// TwinCAT 3 PLC project Rohlik_Expansion
// ProgramVersion: 3.1.4024.0
// libraries:
//   CmpBitmapPool, * (System)
//   Tc2_EtherCAT, * (Beckhoff Automation GmbH)
//   Tc2_IoFunctions, * (Beckhoff Automation GmbH)
//   Tc2_MC2, * (Beckhoff Automation GmbH)
//   Tc2_ModbusSrv, * (Beckhoff Automation GmbH)
//   Tc2_Standard, * (Beckhoff Automation GmbH)
//   Tc2_SUPS, * (Beckhoff Automation GmbH)
//   Tc2_System, * (Beckhoff Automation GmbH)
//   Tc2_Utilities, * (Beckhoff Automation GmbH)
//   Tc3_Module, * (Beckhoff Automation GmbH)
//   Tc3_PackML_V2, * (Beckhoff Automation GmbH)
//   Util, * (System)
//   VisuDialogs, * (System)
// project tree:
//   02DUTs/ E_PMLUserUnitMode.TcDUT (not stored), E_UnitName.TcDUT (not stored), ModuleID.TcDUT, ST_ChangeIntoProduction.TcDUT, ST_UnitInfo.TcDUT (not stored)
//   Ads/ AbortToteRequestParams.TcDUT (not stored), AutostoreControlCommand.TcDUT, BarcodeValidationRequestParams.TcDUT (not stored), BarcodeVerificationResult.TcDUT (not stored), ButtonStatus.TcDUT (not stored), AirPressureStatus.TcDUT (not stored), DigitalInputStatus.TcDUT (not stored), DigitalOutputStatus.TcDUT, EStopStatus.TcDUT, E_SAFETYDOOR.TcDUT, E_SafetyStates.TcDUT (not stored), FB_AirPressure_Subsystem.TcPOU (not stored), FB_HeartBeat_Subsystem.TcPOU (not stored), FB_Light_tower_module.TcPOU (not stored), FB_MachineControl_Subsystem.TcPOU, FB_Safety_Subsystem.TcPOU, FB_Tote_Subsystem.TcPOU, GeneralStatus.TcDUT, HeartbeatParams.TcDUT (not stored), InboundToteParams.TcDUT, InitToteRequestParams.TcDUT (not stored), LightCurtainStatus.TcDUT, MachineCommandStructure.TcDUT (not stored), MachineControlCommand.TcDUT, MachineControlCommand_1.TcDUT, MachineStatus.TcDUT (not stored), MethodCallReturnValue.TcDUT (not stored), ModelIdentifier.TcDUT (not stored), OrderToteCommand.TcDUT (not stored), OutboundToteParams.TcDUT, PerturbToteParams.TcDUT (not stored), SafetyDoorStatus.TcDUT, SafetyStatus.TcDUT (not stored), SensorStatus.TcDUT, StationMode.TcDUT (not stored), ST_BagOpen.TcDUT, ST_LightTower.TcDUT (not stored), SwapToteParams.TcDUT (not stored), ToteData.TcPOU (not stored), UpdateLightTowerParams.TcDUT, UpdateStationModeParams.TcDUT (not stored)
//   Ads/Ads/ BagOpeningStatus.TcPOU, ST_LightTowerAction.TcDUT (not stored)
//   GVLs/ GVL.TcGVL, GVL_SAFETY.TcGVL (not stored), G_HMI.TcGVL, G_IO.TcGVL, ST_Ifm_Qualifier.TcDUT (not stored), ST_Ifm_RX.TcDUT (not stored), ST_Ifm_TX.TcDUT (not stored), ST_IO_16.TcDUT (not stored), ST_SafetyIO.TcDUT (not stored)
//   / EtherCAT_Task.TcTTO, GlobalTextList.TcGTLO, MianTask.TcTTO (not stored), VisualizationManager.TcVMO (not stored), VISU_TASK.TcTTO (not stored)
//   LogTECH/ LogTechControlCmd.TcDUT (not stored), LogTechStatus.TcDUT, LogTechTransferStatus.TcDUT
//   Mian/axis/ AxisHMI_Ex.TcVIS (not stored), E_HomingSteps.TcDUT (not stored), FB_MotionAxis_MC.TcPOU (not stored), MC_HomeAxis.TcPOU (not stored), ST_MotionAxis_MC.TcDUT
//   Mian/DUTs/ BagStatus.TcDUT (not stored), Buffer_roller.TcDUT, E_Condition.TcDUT, E_LoadingStates.TcDUT, E_SampleStates.TcDUT, E_RollerStates.TcDUT (not stored), E_AutoStore_States.TcDUT, E_topic_sample.TcDUT (not stored), E_Transfer.TcDUT (not stored), E_WorkingStates.TcDUT (not stored), FB_DigitalInput.TcPOU (not stored), FB_GPWM.TcPOU (not stored), Inbound.TcDUT, I_Common.TcIO (not stored), OrderToteErrorStatus.TcDUT (not stored), Outbound.TcDUT, Prepare_Date_Time.TcPOU (not stored), Roller.TcDUT (not stored), Roller_x.TcDUT (not stored), Roller_y.TcDUT, ServerityLevelType.TcDUT, ST_Alarm_Hmi.TcDUT (not stored), ST_control_pannel.TcDUT, ST_EVENT.TcDUT (not stored), ST_safetyDoor.TcDUT (not stored), ToteStatus.TcDUT (not stored), ToteSubsystemWorkflowStatus.TcDUT, Valve.TcDUT (not stored)
//   Mian/ FB_Generic.TcPOU (not stored), FB_Machine.TcPOU, FB_mcp.TcPOU (not stored), FB_Sample.TcPOU (not stored), FB_loading_tote.TcPOU (not stored), FB_autoStore.TcPOU, FB_StateMachine.TcPOU, FB_working_tote.TcPOU, FB_Visu.TcPOU (not stored), FB_WriteLog.TcPOU (not stored), MAIN.TcPOU
//   PubSub/ E_Topics.TcDUT, I_PubSubService.TcIO (not stored), I_SubCallback.TcIO (not stored), KeyAndValue.TcDUT, PubSubData.TcDUT (not stored), PubSubService.TcPOU, ST_TracePublish.TcDUT (not stored), SubscriberCell.TcDUT
//   VISUs/ ImagePool.TcIPO (not stored), visu_main.TcVIS (not stored)
//   VISUs/Templates/ visu_autoStore.TcVIS, VIS_TemplateCommand.TcVIS (not stored), VIS_TemplateKeys.TcVIS (not stored), VIS_TemplateMachine.TcVIS (not stored), VIS_TemplatePMLStateModel.TcVIS, VIS_TemplateToProduction.TcVIS (not stored), v_io_autoStore.TcVIS
//   VISUs/VISUs/ Menu.TcVIS (not stored), visu_2sys.TcVIS, visu_loading.TcVIS (not stored), visu_operation.TcVIS, visu_sample.TcVIS (not stored), visu_manual.TcVIS, visu_working1.TcVIS, visu_autoStore1.TcVIS, visu_working2.TcVIS, v_alarm.TcVIS, v_io_loading.TcVIS (not stored), v_io_working1.TcVIS, v_io_working2.TcVIS (not stored)
// real-time tasks:
//   TASK PlcTask: cycle T#4ms, priority 20, ADS port 350
//   TASK EtherCAT_Task: cycle T#2ms, priority 2, ADS port 351
//   TASK VISU_TASK: cycle T#100000us, priority 30, ADS port 352
// motion (NC):
//   TASK NC-Task 1 SAF: cycle T#2ms, priority 4, ADS port 501
//   TASK NC-Task 1 SVB: cycle T#10ms, priority 8, ADS port 511
//   AXIS lift_motor (id 3)
//     Velo: SlowManual=5, FastManual=20
//     PositionAreaControl: Enable=false
//     OtherSettings: AllowMotionCmdToSlave=true
//     encoder EncType=19
//       EncPara: ScaleFactorNumerator=3.333333333333, ScaleFactorDenominator=8388608, Inverse=true, MaxCount=#xffffffff, ReferenceSystem=1
//         SoftEndMinControl: Enable=true, Range=-5
//         SoftEndMaxControl: Enable=true, Range=800
//         Inc: RefSoftSyncMask=#x00800000
//     drive DrvType=16
//       DrvPara: Inverse=true, MaxCount=#xffffffff, DriveControlDWord=#x00020100
//         Analog: TorqueSetpointScale=10, ScaleFactorActTorque=0.1
//         TimeComp: TaskDelayCycles=1
//     controller CtrType=1
//       CtrPara: PriorControlFactor=1
//         PosDiffControl: Enable=false
//         Observer: BandWidth=20
//   AXIS working1_lift_motor (id 4)
//     PositionAreaControl: Enable=false
//     OtherSettings: AllowMotionCmdToSlave=true
//     encoder EncType=19
//       EncPara: ScaleFactorNumerator=5, ScaleFactorDenominator=8388608, Inverse=true, MaxCount=#xffffffff, ReferenceSystem=1
//         SoftEndMinControl: Enable=true, Range=-5
//         SoftEndMaxControl: Enable=true, Range=140
//         Inc: RefSoftSyncMask=#x00800000
//     drive DrvType=16
//       DrvPara: Inverse=true, MaxCount=#xffffffff, DriveControlDWord=#x00020100
//         Analog: TorqueSetpointScale=10, ScaleFactorActTorque=0.1
//         TimeComp: TaskDelayCycles=1
//     controller CtrType=1
//       CtrPara: PriorControlFactor=1
//         PosDiffControl: Enable=false
//         Observer: BandWidth=20
//   AXIS working1_open_bag (id 5)
//     General: UnitName=°
//     Dynamic: Acceleration=75, Deceleration=75, Jerk=112.5
//     Velo: SlowManual=1, FastManual=5, Maximum=300
//     PositionAreaControl: Enable=false
//     OtherSettings: AllowMotionCmdToSlave=true
//     encoder EncType=19
//       EncPara: ScaleFactorNumerator=36, ScaleFactorDenominator=8388608, MaxCount=#xffffffff, ReferenceSystem=1
//         SoftEndMinControl: Enable=true
//         SoftEndMaxControl: Enable=true, Range=56
//         Inc: RefSoftSyncMask=#x00800000
//     drive DrvType=16
//       DrvPara: MaxCount=#xffffffff, DriveControlDWord=#x00020100
//         Analog: TorqueSetpointScale=10, ScaleFactorActTorque=0.1
//         TimeComp: TaskDelayCycles=1
//     controller CtrType=1
//       CtrPara: PriorControlFactor=1
//         PosDiffControl: Enable=false
//         Observer: BandWidth=20
//   AXIS working2_lift_motor (id 1)
//     PositionAreaControl: Enable=false
//     OtherSettings: AllowMotionCmdToSlave=true
//     encoder EncType=19
//       EncPara: ScaleFactorNumerator=5, ScaleFactorDenominator=8388608, Inverse=true, MaxCount=#xffffffff, ReferenceSystem=1
//         SoftEndMinControl: Enable=true, Range=-5
//         SoftEndMaxControl: Enable=true, Range=140
//         Inc: RefSoftSyncMask=#x00800000
//     drive DrvType=16
//       DrvPara: Inverse=true, MaxCount=#xffffffff, DriveControlDWord=#x00020100
//         Analog: TorqueSetpointScale=10, ScaleFactorActTorque=0.1
//         TimeComp: TaskDelayCycles=1
//     controller CtrType=1
//       CtrPara: PriorControlFactor=1
//         PosDiffControl: Enable=false
//         Observer: BandWidth=20
//   AXIS working2_open_bag (id 2)
//     General: UnitName=°
//     Dynamic: Acceleration=75, Deceleration=75, Jerk=112.5
//     Velo: Maximum=300
//     PositionAreaControl: Enable=false
//     OtherSettings: AllowMotionCmdToSlave=true
//     encoder EncType=19
//       EncPara: ScaleFactorNumerator=36, ScaleFactorDenominator=8388608, MaxCount=#xffffffff, ReferenceSystem=1
//         SoftEndMinControl: Enable=true
//         SoftEndMaxControl: Enable=true, Range=56
//         Inc: RefSoftSyncMask=#x00800000
//     drive DrvType=16
//       DrvPara: MaxCount=#xffffffff, DriveControlDWord=#x00020100
//         Analog: TorqueSetpointScale=10, ScaleFactorActTorque=0.1
//         TimeComp: TaskDelayCycles=1
//     controller CtrType=1
//       CtrPara: PriorControlFactor=1
//         PosDiffControl: Enable=false
//         Observer: BandWidth=20
//   AXIS autostore1_transfer (id 6)
//     OtherSettings: AllowMotionCmdToSlave=true
//     encoder EncType=1
//     drive DrvType=5
//       Analog: TorqueSetpointScale=10, ScaleFactorActTorque=0.1
//     controller CtrType=1
//       CtrPara: PriorControlFactor=1
//         Observer: BandWidth=20
//   AXIS autostore1_lift (id 7)
//     OtherSettings: AllowMotionCmdToSlave=true
//     encoder EncType=1
//     drive DrvType=5
//       Analog: TorqueSetpointScale=10, ScaleFactorActTorque=0.1
//     controller CtrType=1
//       CtrPara: PriorControlFactor=1
//         Observer: BandWidth=20
//   AXIS autostore2_transfer (id 8)
//     OtherSettings: AllowMotionCmdToSlave=true
//     encoder EncType=1
//     drive DrvType=5
//       Analog: TorqueSetpointScale=10, ScaleFactorActTorque=0.1
//     controller CtrType=1
//       CtrPara: PriorControlFactor=1
//         Observer: BandWidth=20
//   AXIS autostore2_lift (id 9)
//     OtherSettings: AllowMotionCmdToSlave=true
//     encoder EncType=1
//     drive DrvType=5
//       Analog: TorqueSetpointScale=10, ScaleFactorActTorque=0.1
//     controller CtrType=1
//       CtrPara: PriorControlFactor=1
//         Observer: BandWidth=20
// I/O:
//   DEVICE Device 2 (RT-Ethernet Adapter)
//   DEVICE MCP, AmsNetId 192.168.17.27.4.1
//     Box 1 (CU2508) [CU2508 Ethernet Port]
//     MCP-EK1100 [EK1100 EtherCAT Coupler (2A E-Bus)]
//       DI0 [EL1809 16Ch. Dig. Input 24V, 3ms]
//       DI1 [EL1809 16Ch. Dig. Input 24V, 3ms]
//       DO0 [EL2809 16Ch. Dig. Output 24V, 0.5A]
//       DO1 [EL2809 16Ch. Dig. Output 24V, 0.5A]
//       Term 7 (EL6910) [EL6910, TwinSAFE PLC]
//       SI0 [EL1904, 4 Ch. Safety Input 24V, TwinSAFE]
//         modules: Module 1 (FSOES)
//       SI1 [EL1904, 4 Ch. Safety Input 24V, TwinSAFE]
//         modules: Module 1 (FSOES)
//       SI2 [EL1904, 4 Ch. Safety Input 24V, TwinSAFE]
//         modules: Module 1 (FSOES)
//       SI3 [EL1904, 4 Ch. Safety Input 24V, TwinSAFE]
//         modules: Module 1 (FSOES)
//       SO0 [EL2904, 4 Ch. Safety Output 24V, 0.5A, TwinSAFE]
//         modules: Module 1 (FSOES), Module 2 (DO)
//       SO4 [EL2904, 4 Ch. Safety Output 24V, 0.5A, TwinSAFE]
//         modules: Module 1 (FSOES), Module 2 (DO)
//       Term 50 (EL9410) [EL9410 E-Bus Power Supplier  (Diagnostics)]
//       Term 13 (EL3064) [EL3064 4Ch. Ana. Input 0-10V]
//       SI7 [EL1904, 4 Ch. Safety Input 24V, TwinSAFE]
//         modules: Module 1 (FSOES)
//       SI8 [EL1904, 4 Ch. Safety Input 24V, TwinSAFE]
//         modules: Module 1 (FSOES)
//       SO5 [EL2904, 4 Ch. Safety Output 24V, 0.5A, TwinSAFE]
//         modules: Module 1 (FSOES), Module 2 (DO)
//       SO6 [EL2904, 4 Ch. Safety Output 24V, 0.5A, TwinSAFE]
//         modules: Module 1 (FSOES), Module 2 (DO)
//       Term 14 (EL6631-0010) [EL6631-0010 PROFINET IO Device]
//       Term 15 (EL9011) [EL9011 End Terminal]
//   DEVICE Lift, AmsNetId 192.168.17.27.5.1
//     Box 16 (CU2508) [CU2508 Ethernet Port]
//     Term 17 (EK1100) [EK1100 EtherCAT Coupler (2A E-Bus)]
//       DI2 [EL1809 16Ch. Dig. Input 24V, 3ms]
//       DI3 [EL1809 16Ch. Dig. Input 24V, 3ms]
//       DO2 [EL2809 16Ch. Dig. Output 24V, 0.5A]
//       DO3 [EL2809 16Ch. Dig. Output 24V, 0.5A]
//       SI4 [EL1904, 4 Ch. Safety Input 24V, TwinSAFE]
//         modules: Module 1 (FSOES)
//       SI5 [EL1904, 4 Ch. Safety Input 24V, TwinSAFE]
//         modules: Module 1 (FSOES)
//       SI6 [EL1904, 4 Ch. Safety Input 24V, TwinSAFE]
//         modules: Module 1 (FSOES)
//       SO1 [EL2904, 4 Ch. Safety Output 24V, 0.5A, TwinSAFE]
//         modules: Module 1 (FSOES), Module 2 (DO)
//       Term 10 (EL9011) [EL9011 End Terminal]
//     lift_lift [SV660_1Axis_00915]
//     Box 26 (ifm IO-Link Master AL1332) [ifm IO-Link Master AL1332]
//       modules: Module 1 (IOL_4/4_I/O-Bytes), Module 2 (IOL_4/4_I/O-Bytes), Module 3 (IOL_4/4_I/O-Bytes), Module 4 (IOL_4/4_I/O-Bytes), Module 5 (IOL_4/4_I/O-Bytes), Module 6 (IOL_4/4_I/O-Bytes), Module 7 (IOL_4/4_I/O-Bytes), Module 8 (IOL_4/4_I/O-Bytes)
//   DEVICE Place1, AmsNetId 192.168.17.27.6.1
//     Box 26 (CU2508) [CU2508 Ethernet Port]
//     Term 27 (EK1100) [EK1100 EtherCAT Coupler (2A E-Bus)]
//       DI4 [EL1809 16Ch. Dig. Input 24V, 3ms]
//       DI5 [EL1809 16Ch. Dig. Input 24V, 3ms]
//       DO4 [EL2809 16Ch. Dig. Output 24V, 0.5A]
//       SO2 [EL2904, 4 Ch. Safety Output 24V, 0.5A, TwinSAFE]
//         modules: Module 1 (FSOES), Module 2 (DO)
//       Term 53 (EL9410) [EL9410 E-Bus Power Supplier  (Diagnostics)]
//       DO6 [EL2809 16Ch. Dig. Output 24V, 0.5A]
//       Term 9 (EL9011) [EL9011 End Terminal]
//     place1_lift [SV660_1Axis_00915]
//     place_openbag [SV660_1Axis_00915]
//     Box 36 (ifm IO-Link Master AL1332) [ifm IO-Link Master AL1332]
//       modules: Module 1 (IOL_4/4_I/O-Bytes), Module 2 (IOL_4/4_I/O-Bytes), Module 3 (IOL_4/4_I/O-Bytes), Module 4 (IOL_4/4_I/O-Bytes), Module 5 (IOL_4/4_I/O-Bytes), Module 6 (IOL_4/4_I/O-Bytes), Module 7 (IOL_4/4_I/O-Bytes), Module 8 (IOL_4/4_I/O-Bytes)
//   DEVICE Place2, AmsNetId 192.168.17.27.7.1
//     Box 35 (CU2508) [CU2508 Ethernet Port]
//     Term 36 (EK1100) [EK1100 EtherCAT Coupler (2A E-Bus)]
//       DI6 [EL1809 16Ch. Dig. Input 24V, 3ms]
//       DI7 [EL1809 16Ch. Dig. Input 24V, 3ms]
//       DO5 [EL2809 16Ch. Dig. Output 24V, 0.5A]
//       SO3 [EL2904, 4 Ch. Safety Output 24V, 0.5A, TwinSAFE]
//         modules: Module 1 (FSOES), Module 2 (DO)
//       Term 51 (EL9410) [EL9410 E-Bus Power Supplier  (Diagnostics)]
//       DO7 [EL2809 16Ch. Dig. Output 24V, 0.5A]
//       Term 9 (EL9011) [EL9011 End Terminal]
//     place2_lift [SV660_1Axis_00915]
//     place2_openbag [SV660_1Axis_00915]
//     Box 46 (ifm IO-Link Master AL1332) [ifm IO-Link Master AL1332]
//       modules: Module 1 (IOL_4/4_I/O-Bytes), Module 2 (IOL_4/4_I/O-Bytes), Module 3 (IOL_4/4_I/O-Bytes), Module 4 (IOL_4/4_I/O-Bytes), Module 5 (IOL_4/4_I/O-Bytes), Module 6 (IOL_4/4_I/O-Bytes), Module 7 (IOL_4/4_I/O-Bytes), Module 8 (IOL_4/4_I/O-Bytes)
//   DEVICE Device 1 (EtherCAT Automation Protocol), AmsNetId 192.168.11.159.2.1
// variable links:
//   Lift <-> MCP/MCP-EK1100/Term 7 (EL6910)
//     Term 17 (EK1100)/SI5/Module 1 (FSOES)/RxPDO/FSOE <-> ConnectionInputs/Message_29 TxPDO
//     Term 17 (EK1100)/SI6/Module 1 (FSOES)/RxPDO/FSOE <-> ConnectionInputs/Message_30 TxPDO
//     Term 17 (EK1100)/SI5/Module 1 (FSOES)/TxPDO/FSOE <-> ConnectionOutputs/Message_29 RxPDO
//     Term 17 (EK1100)/SI6/Module 1 (FSOES)/TxPDO/FSOE <-> ConnectionOutputs/Message_30 RxPDO
//   MCP <-> Lift/Term 17 (EK1100)/SI4
//     MCP-EK1100/Term 7 (EL6910)/ConnectionInputs/Message_28 TxPDO <-> Module 1 (FSOES)/RxPDO/FSOE
//     MCP-EK1100/Term 7 (EL6910)/ConnectionOutputs/Message_28 RxPDO <-> Module 1 (FSOES)/TxPDO/FSOE
//   MCP <-> Lift/Term 17 (EK1100)/SO1
//     MCP-EK1100/Term 7 (EL6910)/ConnectionInputs/Message_31 TxPDO <-> Module 1 (FSOES)/RxPDO/FSOE
//     MCP-EK1100/Term 7 (EL6910)/ConnectionOutputs/Message_31 RxPDO <-> Module 1 (FSOES)/TxPDO/FSOE
//   MCP <-> MCP/MCP-EK1100/SI0
//     MCP-EK1100/Term 7 (EL6910)/ConnectionOutputs/Message_22 RxPDO <-> Module 1 (FSOES)/TxPDO/FSOE
//   MCP <-> MCP/MCP-EK1100/SI1
//     MCP-EK1100/Term 7 (EL6910)/ConnectionInputs/Message_23 TxPDO <-> Module 1 (FSOES)/RxPDO/FSOE
//   MCP <-> MCP/MCP-EK1100/SI2
//     MCP-EK1100/Term 7 (EL6910)/ConnectionInputs/Message_24 TxPDO <-> Module 1 (FSOES)/RxPDO/FSOE
//     MCP-EK1100/Term 7 (EL6910)/ConnectionOutputs/Message_24 RxPDO <-> Module 1 (FSOES)/TxPDO/FSOE
//   MCP <-> MCP/MCP-EK1100/SI3
//     MCP-EK1100/Term 7 (EL6910)/ConnectionInputs/Message_27 TxPDO <-> Module 1 (FSOES)/RxPDO/FSOE
//   MCP <-> MCP/MCP-EK1100/SO0
//     MCP-EK1100/Term 7 (EL6910)/ConnectionInputs/Message_26 TxPDO <-> Module 1 (FSOES)/RxPDO/FSOE
//   MCP <-> MCP/MCP-EK1100/SO4
//     MCP-EK1100/Term 7 (EL6910)/ConnectionInputs/Message_36 TxPDO <-> Module 1 (FSOES)/RxPDO/FSOE
//   MCP <-> MCP/MCP-EK1100/SO6
//     MCP-EK1100/Term 7 (EL6910)/ConnectionInputs/Message_72 TxPDO <-> Module 1 (FSOES)/RxPDO/FSOE
//     MCP-EK1100/Term 7 (EL6910)/ConnectionOutputs/Message_72 RxPDO <-> Module 1 (FSOES)/TxPDO/FSOE
//   MCP <-> MCP/MCP-EK1100/Term 7 (EL6910)
//     MCP-EK1100/SI0/Module 1 (FSOES)/RxPDO/FSOE <-> ConnectionInputs/Message_22 TxPDO
//     MCP-EK1100/SI1/Module 1 (FSOES)/TxPDO/FSOE <-> ConnectionOutputs/Message_23 RxPDO
//     MCP-EK1100/SI3/Module 1 (FSOES)/TxPDO/FSOE <-> ConnectionOutputs/Message_27 RxPDO
//     MCP-EK1100/SO0/Module 1 (FSOES)/TxPDO/FSOE <-> ConnectionOutputs/Message_26 RxPDO
//     MCP-EK1100/SO4/Module 1 (FSOES)/TxPDO/FSOE <-> ConnectionOutputs/Message_36 RxPDO
//     MCP-EK1100/SO5/Module 1 (FSOES)/TxPDO/FSOE <-> ConnectionOutputs/Message_71 RxPDO
//     MCP-EK1100/SO5/Module 1 (FSOES)/RxPDO/FSOE <-> ConnectionInputs/Message_71 TxPDO
//   MCP <-> Place2/Term 36 (EK1100)/SO3
//     MCP-EK1100/Term 7 (EL6910)/ConnectionInputs/Message_33 TxPDO <-> Module 1 (FSOES)/RxPDO/FSOE
//     MCP-EK1100/Term 7 (EL6910)/ConnectionOutputs/Message_33 RxPDO <-> Module 1 (FSOES)/TxPDO/FSOE
//   Place1 <-> MCP/MCP-EK1100/Term 7 (EL6910)
//     Term 27 (EK1100)/SO2/Module 1 (FSOES)/RxPDO/FSOE <-> ConnectionInputs/Message_32 TxPDO
//     Term 27 (EK1100)/SO2/Module 1 (FSOES)/TxPDO/FSOE <-> ConnectionOutputs/Message_32 RxPDO
//   NC-Task 1 SAF/Axes/lift_motor <-> Lift/lift_lift
//     Drive/Inputs/In/nDataIn1 <-> Inputs/Following error actual value
//     Drive/Inputs/In/nDataIn3[0] <-> Inputs/Torque actual value
//     Drive/Inputs/In/nDcOutputTime <-> InfoData/DcOutputShift
//     Drive/Inputs/In/nState1 <-> Inputs/Statusword
//     Drive/Inputs/In/nState2 <-> Inputs/Statusword @bit 8
//     Drive/Inputs/In/nState4 @bit 1 <-> WcState/InputToggle
//     Drive/Inputs/In/nState4 <-> WcState/WcState
//     Drive/Outputs/Out/nCtrl1 <-> Outputs/Controlword
//     Drive/Outputs/Out/nCtrl2 <-> Outputs/Controlword @bit 8
//     Drive/Outputs/Out/nDataOut1 <-> Outputs/Target position
//     Enc/Inputs/In/nDataIn1 <-> Inputs/Position actual value
//     Enc/Inputs/In/nDataIn3 <-> Inputs/Touch probe pos1 pos value
//     Enc/Inputs/In/nDataIn5 <-> Inputs/Touch probe pos2 pos value
//     Enc/Inputs/In/nDcInputTime <-> InfoData/DcInputShift
//     Enc/Inputs/In/nState4 @bit 1 <-> WcState/InputToggle
//     Enc/Inputs/In/nState4 <-> WcState/WcState
//     Enc/Inputs/In/nState5 <-> Inputs/Touch probe status
//     Enc/Inputs/In/nState6 <-> Inputs/Touch probe status @bit 8
//     Enc/Outputs/Out/nCtrl5 <-> Outputs/Touch probe function
//     Enc/Outputs/Out/nCtrl6 <-> Outputs/Touch probe function @bit 8
//   NC-Task 1 SAF/Axes/working1_lift_motor <-> Place1/place1_lift
//     Drive/Inputs/In/nDataIn1 <-> Inputs/Following error actual value
//     Drive/Inputs/In/nDataIn3[0] <-> Inputs/Torque actual value
//     Drive/Inputs/In/nDcOutputTime <-> InfoData/DcOutputShift
//     Drive/Inputs/In/nState1 <-> Inputs/Statusword
//     Drive/Inputs/In/nState2 <-> Inputs/Statusword @bit 8
//     Drive/Inputs/In/nState4 @bit 1 <-> WcState/InputToggle
//     Drive/Inputs/In/nState4 <-> WcState/WcState
//     Drive/Outputs/Out/nCtrl1 <-> Outputs/Controlword
//     Drive/Outputs/Out/nCtrl2 <-> Outputs/Controlword @bit 8
//     Drive/Outputs/Out/nDataOut1 <-> Outputs/Target position
//     Enc/Inputs/In/nDataIn1 <-> Inputs/Position actual value
//     Enc/Inputs/In/nDataIn3 <-> Inputs/Touch probe pos1 pos value
//     Enc/Inputs/In/nDataIn5 <-> Inputs/Touch probe pos2 pos value
//     Enc/Inputs/In/nDcInputTime <-> InfoData/DcInputShift
//     Enc/Inputs/In/nState4 @bit 1 <-> WcState/InputToggle
//     Enc/Inputs/In/nState4 <-> WcState/WcState
//     Enc/Inputs/In/nState5 <-> Inputs/Touch probe status
//     Enc/Inputs/In/nState6 <-> Inputs/Touch probe status @bit 8
//     Enc/Outputs/Out/nCtrl5 <-> Outputs/Touch probe function
//     Enc/Outputs/Out/nCtrl6 <-> Outputs/Touch probe function @bit 8
//   NC-Task 1 SAF/Axes/working1_open_bag <-> Place1/place_openbag
//     Drive/Inputs/In/nDataIn1 <-> Inputs/Following error actual value
//     Drive/Inputs/In/nDataIn3[0] <-> Inputs/Torque actual value
//     Drive/Inputs/In/nDcOutputTime <-> InfoData/DcOutputShift
//     Drive/Inputs/In/nState1 <-> Inputs/Statusword
//     Drive/Inputs/In/nState2 <-> Inputs/Statusword @bit 8
//     Drive/Inputs/In/nState4 @bit 1 <-> WcState/InputToggle
//     Drive/Inputs/In/nState4 <-> WcState/WcState
//     Drive/Outputs/Out/nCtrl1 <-> Outputs/Controlword
//     Drive/Outputs/Out/nCtrl2 <-> Outputs/Controlword @bit 8
//     Drive/Outputs/Out/nDataOut1 <-> Outputs/Target position
//     Enc/Inputs/In/nDataIn1 <-> Inputs/Position actual value
//     Enc/Inputs/In/nDataIn3 <-> Inputs/Touch probe pos1 pos value
//     Enc/Inputs/In/nDataIn5 <-> Inputs/Touch probe pos2 pos value
//     Enc/Inputs/In/nDcInputTime <-> InfoData/DcInputShift
//     Enc/Inputs/In/nState4 @bit 1 <-> WcState/InputToggle
//     Enc/Inputs/In/nState4 <-> WcState/WcState
//     Enc/Inputs/In/nState5 <-> Inputs/Touch probe status
//     Enc/Inputs/In/nState6 <-> Inputs/Touch probe status @bit 8
//     Enc/Outputs/Out/nCtrl5 <-> Outputs/Touch probe function
//     Enc/Outputs/Out/nCtrl6 <-> Outputs/Touch probe function @bit 8
//   NC-Task 1 SAF/Axes/working2_lift_motor <-> Place2/place2_lift
//     Drive/Inputs/In/nDataIn1 <-> Inputs/Following error actual value
//     Drive/Inputs/In/nDataIn3[0] <-> Inputs/Torque actual value
//     Drive/Inputs/In/nDcOutputTime <-> InfoData/DcOutputShift
//     Drive/Inputs/In/nState1 <-> Inputs/Statusword
//     Drive/Inputs/In/nState2 <-> Inputs/Statusword @bit 8
//     Drive/Inputs/In/nState4 @bit 1 <-> WcState/InputToggle
//     Drive/Inputs/In/nState4 <-> WcState/WcState
//     Drive/Outputs/Out/nCtrl1 <-> Outputs/Controlword
//     Drive/Outputs/Out/nCtrl2 <-> Outputs/Controlword @bit 8
//     Drive/Outputs/Out/nDataOut1 <-> Outputs/Target position
//     Enc/Inputs/In/nDataIn1 <-> Inputs/Position actual value
//     Enc/Inputs/In/nDataIn3 <-> Inputs/Touch probe pos1 pos value
//     Enc/Inputs/In/nDataIn5 <-> Inputs/Touch probe pos2 pos value
//     Enc/Inputs/In/nDcInputTime <-> InfoData/DcInputShift
//     Enc/Inputs/In/nState4 @bit 1 <-> WcState/InputToggle
//     Enc/Inputs/In/nState4 <-> WcState/WcState
//     Enc/Inputs/In/nState5 <-> Inputs/Touch probe status
//     Enc/Inputs/In/nState6 <-> Inputs/Touch probe status @bit 8
//     Enc/Outputs/Out/nCtrl5 <-> Outputs/Touch probe function
//     Enc/Outputs/Out/nCtrl6 <-> Outputs/Touch probe function @bit 8
//   NC-Task 1 SAF/Axes/working2_open_bag <-> Place2/place2_openbag
//     Drive/Inputs/In/nDataIn1 <-> Inputs/Following error actual value
//     Drive/Inputs/In/nDataIn3[0] <-> Inputs/Torque actual value
//     Drive/Inputs/In/nDcOutputTime <-> InfoData/DcOutputShift
//     Drive/Inputs/In/nState1 <-> Inputs/Statusword
//     Drive/Inputs/In/nState2 <-> Inputs/Statusword @bit 8
//     Drive/Inputs/In/nState4 @bit 1 <-> WcState/InputToggle
//     Drive/Inputs/In/nState4 <-> WcState/WcState
//     Drive/Outputs/Out/nCtrl1 <-> Outputs/Controlword
//     Drive/Outputs/Out/nCtrl2 <-> Outputs/Controlword @bit 8
//     Drive/Outputs/Out/nDataOut1 <-> Outputs/Target position
//     Enc/Inputs/In/nDataIn1 <-> Inputs/Position actual value
//     Enc/Inputs/In/nDataIn3 <-> Inputs/Touch probe pos1 pos value
//     Enc/Inputs/In/nDataIn5 <-> Inputs/Touch probe pos2 pos value
//     Enc/Inputs/In/nDcInputTime <-> InfoData/DcInputShift
//     Enc/Inputs/In/nState4 @bit 1 <-> WcState/InputToggle
//     Enc/Inputs/In/nState4 <-> WcState/WcState
//     Enc/Inputs/In/nState5 <-> Inputs/Touch probe status
//     Enc/Inputs/In/nState6 <-> Inputs/Touch probe status @bit 8
//     Enc/Outputs/Out/nCtrl5 <-> Outputs/Touch probe function
//     Enc/Outputs/Out/nCtrl6 <-> Outputs/Touch probe function @bit 8
//   Rohlik_Expansion/Rohlik_Expansion Instance <-> Device 1 (EtherCAT Automation Protocol)
//     MianTask Inputs/G_IO.devState_Device1 <-> Inputs/DevState
//   Rohlik_Expansion/Rohlik_Expansion Instance <-> Lift
//     MianTask Inputs/G_IO.wcState_lift <-> Inputs/Frm0WcState
//   Rohlik_Expansion/Rohlik_Expansion Instance <-> Lift/Box 26 (ifm IO-Link Master AL1332)
//     MianTask Inputs/G_IO.arIOLinkQualifier_Lift/CH[{0..7}] <-> TxPDO IO-Link Port Qualifier/Qualifier of IO-Link Ch.{1..8}  (8 links)
//     MianTask Inputs/G_IO.arIOLinkTx_Lift[0]/InputByte[0] <-> Module 1 (IOL_4/4_I/O-Bytes)/TxPDO/input byte 0
//     MianTask Inputs/G_IO.arIOLinkTx_Lift[0]/InputByte[1] <-> Module 1 (IOL_4/4_I/O-Bytes)/TxPDO/input byte 1
//     MianTask Inputs/G_IO.arIOLinkTx_Lift[0]/InputByte[2] <-> Module 1 (IOL_4/4_I/O-Bytes)/TxPDO/input byte 2
//     MianTask Inputs/G_IO.arIOLinkTx_Lift[0]/InputByte[3] <-> Module 1 (IOL_4/4_I/O-Bytes)/TxPDO/input byte 3
//     MianTask Inputs/G_IO.arIOLinkTx_Lift[1]/InputByte[0] <-> Module 2 (IOL_4/4_I/O-Bytes)/TxPDO/input byte 0
//     MianTask Inputs/G_IO.arIOLinkTx_Lift[1]/InputByte[1] <-> Module 2 (IOL_4/4_I/O-Bytes)/TxPDO/input byte 1
//     MianTask Inputs/G_IO.arIOLinkTx_Lift[1]/InputByte[2] <-> Module 2 (IOL_4/4_I/O-Bytes)/TxPDO/input byte 2
//     MianTask Inputs/G_IO.arIOLinkTx_Lift[1]/InputByte[3] <-> Module 2 (IOL_4/4_I/O-Bytes)/TxPDO/input byte 3
//     MianTask Inputs/G_IO.arIOLinkTx_Lift[2]/InputByte[0] <-> Module 3 (IOL_4/4_I/O-Bytes)/TxPDO/input byte 0
//     MianTask Inputs/G_IO.arIOLinkTx_Lift[2]/InputByte[1] <-> Module 3 (IOL_4/4_I/O-Bytes)/TxPDO/input byte 1
//     MianTask Inputs/G_IO.arIOLinkTx_Lift[2]/InputByte[2] <-> Module 3 (IOL_4/4_I/O-Bytes)/TxPDO/input byte 2
//     MianTask Inputs/G_IO.arIOLinkTx_Lift[2]/InputByte[3] <-> Module 3 (IOL_4/4_I/O-Bytes)/TxPDO/input byte 3
//     MianTask Inputs/G_IO.arIOLinkTx_Lift[3]/InputByte[0] <-> Module 4 (IOL_4/4_I/O-Bytes)/TxPDO/input byte 0
//     MianTask Inputs/G_IO.arIOLinkTx_Lift[3]/InputByte[1] <-> Module 4 (IOL_4/4_I/O-Bytes)/TxPDO/input byte 1
//     MianTask Inputs/G_IO.arIOLinkTx_Lift[3]/InputByte[2] <-> Module 4 (IOL_4/4_I/O-Bytes)/TxPDO/input byte 2
//     MianTask Inputs/G_IO.arIOLinkTx_Lift[3]/InputByte[3] <-> Module 4 (IOL_4/4_I/O-Bytes)/TxPDO/input byte 3
//     MianTask Inputs/G_IO.arIOLinkTx_Lift[4]/InputByte[0] <-> Module 5 (IOL_4/4_I/O-Bytes)/TxPDO/input byte 0
//     MianTask Inputs/G_IO.arIOLinkTx_Lift[4]/InputByte[1] <-> Module 5 (IOL_4/4_I/O-Bytes)/TxPDO/input byte 1
//     MianTask Inputs/G_IO.arIOLinkTx_Lift[4]/InputByte[2] <-> Module 5 (IOL_4/4_I/O-Bytes)/TxPDO/input byte 2
//     MianTask Inputs/G_IO.arIOLinkTx_Lift[4]/InputByte[3] <-> Module 5 (IOL_4/4_I/O-Bytes)/TxPDO/input byte 3
//     MianTask Inputs/G_IO.arIOLinkTx_Lift[5]/InputByte[0] <-> Module 6 (IOL_4/4_I/O-Bytes)/TxPDO/input byte 0
//     MianTask Inputs/G_IO.arIOLinkTx_Lift[5]/InputByte[1] <-> Module 6 (IOL_4/4_I/O-Bytes)/TxPDO/input byte 1
//     MianTask Inputs/G_IO.arIOLinkTx_Lift[5]/InputByte[2] <-> Module 6 (IOL_4/4_I/O-Bytes)/TxPDO/input byte 2
//     MianTask Inputs/G_IO.arIOLinkTx_Lift[5]/InputByte[3] <-> Module 6 (IOL_4/4_I/O-Bytes)/TxPDO/input byte 3
//     MianTask Inputs/G_IO.arIOLinkTx_Lift[6]/InputByte[0] <-> Module 7 (IOL_4/4_I/O-Bytes)/TxPDO/input byte 0
//     MianTask Inputs/G_IO.arIOLinkTx_Lift[6]/InputByte[1] <-> Module 7 (IOL_4/4_I/O-Bytes)/TxPDO/input byte 1
//     MianTask Inputs/G_IO.arIOLinkTx_Lift[6]/InputByte[2] <-> Module 7 (IOL_4/4_I/O-Bytes)/TxPDO/input byte 2
//     MianTask Inputs/G_IO.arIOLinkTx_Lift[6]/InputByte[3] <-> Module 7 (IOL_4/4_I/O-Bytes)/TxPDO/input byte 3
//     MianTask Inputs/G_IO.arIOLinkTx_Lift[7]/InputByte[0] <-> Module 8 (IOL_4/4_I/O-Bytes)/TxPDO/input byte 0
//     MianTask Inputs/G_IO.arIOLinkTx_Lift[7]/InputByte[1] <-> Module 8 (IOL_4/4_I/O-Bytes)/TxPDO/input byte 1
//     MianTask Inputs/G_IO.arIOLinkTx_Lift[7]/InputByte[2] <-> Module 8 (IOL_4/4_I/O-Bytes)/TxPDO/input byte 2
//     MianTask Inputs/G_IO.arIOLinkTx_Lift[7]/InputByte[3] <-> Module 8 (IOL_4/4_I/O-Bytes)/TxPDO/input byte 3
//     MianTask Outputs/G_IO.arIOLinkRx_Lift[0]/OutputByte[0] <-> Module 1 (IOL_4/4_I/O-Bytes)/RxPDO/output byte 0
//     MianTask Outputs/G_IO.arIOLinkRx_Lift[0]/OutputByte[1] <-> Module 1 (IOL_4/4_I/O-Bytes)/RxPDO/output byte 1
//     MianTask Outputs/G_IO.arIOLinkRx_Lift[0]/OutputByte[2] <-> Module 1 (IOL_4/4_I/O-Bytes)/RxPDO/output byte 2
//     MianTask Outputs/G_IO.arIOLinkRx_Lift[0]/OutputByte[3] <-> Module 1 (IOL_4/4_I/O-Bytes)/RxPDO/output byte 3
//     MianTask Outputs/G_IO.arIOLinkRx_Lift[1]/OutputByte[0] <-> Module 2 (IOL_4/4_I/O-Bytes)/RxPDO/output byte 0
//     MianTask Outputs/G_IO.arIOLinkRx_Lift[1]/OutputByte[1] <-> Module 2 (IOL_4/4_I/O-Bytes)/RxPDO/output byte 1
//     MianTask Outputs/G_IO.arIOLinkRx_Lift[1]/OutputByte[2] <-> Module 2 (IOL_4/4_I/O-Bytes)/RxPDO/output byte 2
//     MianTask Outputs/G_IO.arIOLinkRx_Lift[1]/OutputByte[3] <-> Module 2 (IOL_4/4_I/O-Bytes)/RxPDO/output byte 3
//     MianTask Outputs/G_IO.arIOLinkRx_Lift[2]/OutputByte[0] <-> Module 3 (IOL_4/4_I/O-Bytes)/RxPDO/output byte 0
//     MianTask Outputs/G_IO.arIOLinkRx_Lift[2]/OutputByte[1] <-> Module 3 (IOL_4/4_I/O-Bytes)/RxPDO/output byte 1
//     MianTask Outputs/G_IO.arIOLinkRx_Lift[2]/OutputByte[2] <-> Module 3 (IOL_4/4_I/O-Bytes)/RxPDO/output byte 2
//     MianTask Outputs/G_IO.arIOLinkRx_Lift[2]/OutputByte[3] <-> Module 3 (IOL_4/4_I/O-Bytes)/RxPDO/output byte 3
//     MianTask Outputs/G_IO.arIOLinkRx_Lift[3]/OutputByte[0] <-> Module 4 (IOL_4/4_I/O-Bytes)/RxPDO/output byte 0
//     MianTask Outputs/G_IO.arIOLinkRx_Lift[3]/OutputByte[1] <-> Module 4 (IOL_4/4_I/O-Bytes)/RxPDO/output byte 1
//     MianTask Outputs/G_IO.arIOLinkRx_Lift[3]/OutputByte[2] <-> Module 4 (IOL_4/4_I/O-Bytes)/RxPDO/output byte 2
//     MianTask Outputs/G_IO.arIOLinkRx_Lift[3]/OutputByte[3] <-> Module 4 (IOL_4/4_I/O-Bytes)/RxPDO/output byte 3
//     MianTask Outputs/G_IO.arIOLinkRx_Lift[4]/OutputByte[0] <-> Module 5 (IOL_4/4_I/O-Bytes)/RxPDO/output byte 0
//     MianTask Outputs/G_IO.arIOLinkRx_Lift[4]/OutputByte[1] <-> Module 5 (IOL_4/4_I/O-Bytes)/RxPDO/output byte 1
//     MianTask Outputs/G_IO.arIOLinkRx_Lift[4]/OutputByte[2] <-> Module 5 (IOL_4/4_I/O-Bytes)/RxPDO/output byte 2
//     MianTask Outputs/G_IO.arIOLinkRx_Lift[4]/OutputByte[3] <-> Module 5 (IOL_4/4_I/O-Bytes)/RxPDO/output byte 3
//     MianTask Outputs/G_IO.arIOLinkRx_Lift[5]/OutputByte[0] <-> Module 6 (IOL_4/4_I/O-Bytes)/RxPDO/output byte 0
//     MianTask Outputs/G_IO.arIOLinkRx_Lift[5]/OutputByte[1] <-> Module 6 (IOL_4/4_I/O-Bytes)/RxPDO/output byte 1
//     MianTask Outputs/G_IO.arIOLinkRx_Lift[5]/OutputByte[2] <-> Module 6 (IOL_4/4_I/O-Bytes)/RxPDO/output byte 2
//     MianTask Outputs/G_IO.arIOLinkRx_Lift[5]/OutputByte[3] <-> Module 6 (IOL_4/4_I/O-Bytes)/RxPDO/output byte 3
//     MianTask Outputs/G_IO.arIOLinkRx_Lift[6]/OutputByte[0] <-> Module 7 (IOL_4/4_I/O-Bytes)/RxPDO/output byte 0
//     MianTask Outputs/G_IO.arIOLinkRx_Lift[6]/OutputByte[1] <-> Module 7 (IOL_4/4_I/O-Bytes)/RxPDO/output byte 1
//     MianTask Outputs/G_IO.arIOLinkRx_Lift[6]/OutputByte[2] <-> Module 7 (IOL_4/4_I/O-Bytes)/RxPDO/output byte 2
//     MianTask Outputs/G_IO.arIOLinkRx_Lift[6]/OutputByte[3] <-> Module 7 (IOL_4/4_I/O-Bytes)/RxPDO/output byte 3
//     MianTask Outputs/G_IO.arIOLinkRx_Lift[7]/OutputByte[0] <-> Module 8 (IOL_4/4_I/O-Bytes)/RxPDO/output byte 0
//     MianTask Outputs/G_IO.arIOLinkRx_Lift[7]/OutputByte[1] <-> Module 8 (IOL_4/4_I/O-Bytes)/RxPDO/output byte 1
//     MianTask Outputs/G_IO.arIOLinkRx_Lift[7]/OutputByte[2] <-> Module 8 (IOL_4/4_I/O-Bytes)/RxPDO/output byte 2
//     MianTask Outputs/G_IO.arIOLinkRx_Lift[7]/OutputByte[3] <-> Module 8 (IOL_4/4_I/O-Bytes)/RxPDO/output byte 3
//   Rohlik_Expansion/Rohlik_Expansion Instance <-> Lift/Term 17 (EK1100)/DI2
//     MianTask Inputs/G_IO.arDI[2]/Ch[{0..15}] <-> Channel {1..16}/Input  (16 links)
//   Rohlik_Expansion/Rohlik_Expansion Instance <-> Lift/Term 17 (EK1100)/DI3
//     MianTask Inputs/G_IO.arDI[3]/Ch[{0..15}] <-> Channel {1..16}/Input  (16 links)
//   Rohlik_Expansion/Rohlik_Expansion Instance <-> Lift/Term 17 (EK1100)/DO2
//     MianTask Outputs/G_IO.arDO[2]/Ch[{0..15}] <-> Channel {1..16}/Output  (16 links)
//   Rohlik_Expansion/Rohlik_Expansion Instance <-> Lift/Term 17 (EK1100)/DO3
//     MianTask Outputs/G_IO.arDO[3]/Ch[{0..15}] <-> Channel {1..16}/Output  (16 links)
//   Rohlik_Expansion/Rohlik_Expansion Instance <-> Lift/Term 17 (EK1100)/SI4
//     MianTask Inputs/G_IO.arSI[4]/Ch[{1..4}] <-> Module 1 (FSOES)/TxPDO/FSOE/InputChannel{1..4}  (4 links)
//   Rohlik_Expansion/Rohlik_Expansion Instance <-> Lift/Term 17 (EK1100)/SI5
//     MianTask Inputs/G_IO.arSI[5]/Ch[{1..4}] <-> Module 1 (FSOES)/TxPDO/FSOE/InputChannel{1..4}  (4 links)
//   Rohlik_Expansion/Rohlik_Expansion Instance <-> Lift/Term 17 (EK1100)/SI6
//     MianTask Inputs/G_IO.arSI[6]/Ch[{1..4}] <-> Module 1 (FSOES)/TxPDO/FSOE/InputChannel{1..4}  (4 links)
//   Rohlik_Expansion/Rohlik_Expansion Instance <-> MCP
//     MianTask Inputs/G_IO.wcState_mcp <-> Inputs/Frm0WcState
//   Rohlik_Expansion/Rohlik_Expansion Instance <-> MCP/MCP-EK1100/DI0
//     MianTask Inputs/G_IO.arDI[0]/Ch[{0..15}] <-> Channel {1..16}/Input  (16 links)
//   Rohlik_Expansion/Rohlik_Expansion Instance <-> MCP/MCP-EK1100/DI1
//     MianTask Inputs/G_IO.arDI[1]/Ch[{0..15}] <-> Channel {1..16}/Input  (16 links)
//   Rohlik_Expansion/Rohlik_Expansion Instance <-> MCP/MCP-EK1100/DO0
//     MianTask Outputs/G_IO.arDO[0]/Ch[{0..15}] <-> Channel {1..16}/Output  (16 links)
//   Rohlik_Expansion/Rohlik_Expansion Instance <-> MCP/MCP-EK1100/DO1
//     MianTask Outputs/G_IO.arDO[1]/Ch[{0..15}] <-> Channel {1..16}/Output  (16 links)
//   Rohlik_Expansion/Rohlik_Expansion Instance <-> MCP/MCP-EK1100/SI0
//     MianTask Inputs/G_IO.arSI[0]/Ch[{1..4}] <-> Module 1 (FSOES)/TxPDO/FSOE/InputChannel{1..4}  (4 links)
//   Rohlik_Expansion/Rohlik_Expansion Instance <-> MCP/MCP-EK1100/SI1
//     MianTask Inputs/G_IO.arSI[1]/Ch[{1..4}] <-> Module 1 (FSOES)/TxPDO/FSOE/InputChannel{1..4}  (4 links)
//   Rohlik_Expansion/Rohlik_Expansion Instance <-> MCP/MCP-EK1100/SI2
//     MianTask Inputs/G_IO.arSI[2]/Ch[{1..4}] <-> Module 1 (FSOES)/TxPDO/FSOE/InputChannel{1..4}  (4 links)
//   Rohlik_Expansion/Rohlik_Expansion Instance <-> MCP/MCP-EK1100/SI3
//     MianTask Inputs/G_IO.arSI[3]/Ch[{1..4}] <-> Module 1 (FSOES)/TxPDO/FSOE/InputChannel{1..4}  (4 links)
//   Rohlik_Expansion/Rohlik_Expansion Instance <-> MCP/MCP-EK1100/SI7
//     MianTask Inputs/G_IO.arSI[7]/Ch[{1..4}] <-> Module 1 (FSOES)/TxPDO/FSOE/InputChannel{1..4}  (4 links)
//   Rohlik_Expansion/Rohlik_Expansion Instance <-> MCP/MCP-EK1100/SI8
//     MianTask Inputs/G_IO.arSI[8]/Ch[{1..4}] <-> Module 1 (FSOES)/TxPDO/FSOE/InputChannel{1..4}  (4 links)
//   Rohlik_Expansion/Rohlik_Expansion Instance <-> MCP/MCP-EK1100/Term 13 (EL3064)
//     MianTask Inputs/GVL.iAng_AirFlow_left <-> AI Standard Channel 3/Value
//     MianTask Inputs/GVL.iAng_AirFlow_right <-> AI Standard Channel 4/Value
//     MianTask Inputs/GVL.iAng_airPress_left <-> AI Standard Channel 1/Value
//     MianTask Inputs/GVL.iAng_airPress_right <-> AI Standard Channel 2/Value
//   Rohlik_Expansion/Rohlik_Expansion Instance <-> MCP/MCP-EK1100/Term 7 (EL6910)
//     MianTask Inputs/GVL_SAFETY.Lift_STO <-> StandardInputs/Standard Out Var 42
//     MianTask Inputs/GVL_SAFETY.Place1_STO <-> StandardInputs/Standard Out Var 43
//     MianTask Inputs/GVL_SAFETY.Place2_STO <-> StandardInputs/Standard Out Var 44
//     MianTask Inputs/GVL_SAFETY.SO0_0 <-> StandardInputs/Standard Out Var 45
//     MianTask Inputs/GVL_SAFETY.SO0_1 <-> StandardInputs/Standard Out Var 47
//     MianTask Inputs/GVL_SAFETY.SO0_2 <-> StandardInputs/Standard Out Var 46
//     MianTask Inputs/GVL_SAFETY.SO0_3 <-> StandardInputs/Standard Out Var 48
//     MianTask Inputs/GVL_SAFETY.SO1_0 <-> StandardInputs/Standard Out Var 42
//     MianTask Inputs/GVL_SAFETY.SO1_1 <-> StandardInputs/Standard Out Var 43
//     MianTask Inputs/GVL_SAFETY.SO1_2 <-> StandardInputs/Standard Out Var 44
//     MianTask Inputs/GVL_SAFETY.SO2_0 <-> StandardInputs/Standard Out Var 42
//     MianTask Inputs/GVL_SAFETY.SO2_1 <-> StandardInputs/Standard Out Var 43
//     MianTask Inputs/GVL_SAFETY.SO2_2 <-> StandardInputs/Standard Out Var 44
//     MianTask Inputs/GVL_SAFETY.SO3_0 <-> StandardInputs/Standard Out Var 42
//     MianTask Inputs/GVL_SAFETY.SO3_1 <-> StandardInputs/Standard Out Var 43
//     MianTask Inputs/GVL_SAFETY.SO3_2 <-> StandardInputs/Standard Out Var 44
//     MianTask Inputs/GVL_SAFETY.SO4_0 <-> StandardInputs/Standard Out Var 59
//     MianTask Inputs/GVL_SAFETY.SO4_1 <-> StandardInputs/Standard Out Var 60
//     MianTask Inputs/GVL_SAFETY.bAirDump1 <-> StandardInputs/Standard Out Var 74
//     MianTask Inputs/GVL_SAFETY.bAirDump2 <-> StandardInputs/Standard Out Var 75
//     MianTask Inputs/GVL_SAFETY.b_ComError <-> StandardInputs/Standard Out Var 18
//     MianTask Inputs/GVL_SAFETY.b_FBerror <-> StandardInputs/Standard Out Var 19
//     MianTask Inputs/GVL_SAFETY.robot1_STO_EAS <-> StandardInputs/Standard Out Var 47
//     MianTask Inputs/GVL_SAFETY.robot2_STO_EAS <-> StandardInputs/Standard Out Var 48
//     MianTask Inputs/GVL_SAFETY.robot1_STO_EES <-> StandardInputs/Standard Out Var 45
//     MianTask Inputs/GVL_SAFETY.robot2_STO_EES <-> StandardInputs/Standard Out Var 46
//     MianTask Outputs/GVL_SAFETY.bLeftDoorUnlock_Request <-> StandardOutputs/Standard In Var 34
//     MianTask Outputs/GVL_SAFETY.bRightDoorUnlock_Request <-> StandardOutputs/Standard In Var 35
//     MianTask Outputs/GVL_SAFETY.bSafetyReset_airDump <-> StandardOutputs/Standard In Var 73
//     MianTask Outputs/GVL_SAFETY.bSafetyRestart_left <-> StandardOutputs/Standard In Var 65
//     MianTask Outputs/GVL_SAFETY.bSafetyRestart_right <-> StandardOutputs/Standard In Var 66
//     MianTask Outputs/GVL_SAFETY.b_EStopRestart <-> StandardOutputs/Standard In Var 16
//     MianTask Outputs/GVL_SAFETY.b_ErrorAck <-> StandardOutputs/Standard In Var 15
//     MianTask Outputs/GVL_SAFETY.b_GroupRun <-> StandardOutputs/Standard In Var 14
//   Rohlik_Expansion/Rohlik_Expansion Instance <-> Place1
//     MianTask Inputs/G_IO.wcState_place1 <-> Inputs/Frm0WcState
//   Rohlik_Expansion/Rohlik_Expansion Instance <-> Place1/Box 36 (ifm IO-Link Master AL1332)
//     MianTask Inputs/G_IO.arIOLinkQualifier_Place1/CH[{0..7}] <-> TxPDO IO-Link Port Qualifier/Qualifier of IO-Link Ch.{1..8}  (8 links)
//     MianTask Inputs/G_IO.arIOLinkTx_Place1[0]/InputByte[0] <-> Module 1 (IOL_4/4_I/O-Bytes)/TxPDO/input byte 0
//     MianTask Inputs/G_IO.arIOLinkTx_Place1[0]/InputByte[1] <-> Module 1 (IOL_4/4_I/O-Bytes)/TxPDO/input byte 1
//     MianTask Inputs/G_IO.arIOLinkTx_Place1[0]/InputByte[2] <-> Module 1 (IOL_4/4_I/O-Bytes)/TxPDO/input byte 2
//     MianTask Inputs/G_IO.arIOLinkTx_Place1[0]/InputByte[3] <-> Module 1 (IOL_4/4_I/O-Bytes)/TxPDO/input byte 3
//     MianTask Inputs/G_IO.arIOLinkTx_Place1[1]/InputByte[0] <-> Module 2 (IOL_4/4_I/O-Bytes)/TxPDO/input byte 0
//     MianTask Inputs/G_IO.arIOLinkTx_Place1[1]/InputByte[1] <-> Module 2 (IOL_4/4_I/O-Bytes)/TxPDO/input byte 1
//     MianTask Inputs/G_IO.arIOLinkTx_Place1[1]/InputByte[2] <-> Module 2 (IOL_4/4_I/O-Bytes)/TxPDO/input byte 2
//     MianTask Inputs/G_IO.arIOLinkTx_Place1[1]/InputByte[3] <-> Module 2 (IOL_4/4_I/O-Bytes)/TxPDO/input byte 3
//     MianTask Inputs/G_IO.arIOLinkTx_Place1[2]/InputByte[0] <-> Module 3 (IOL_4/4_I/O-Bytes)/TxPDO/input byte 0
//     MianTask Inputs/G_IO.arIOLinkTx_Place1[2]/InputByte[1] <-> Module 3 (IOL_4/4_I/O-Bytes)/TxPDO/input byte 1
//     MianTask Inputs/G_IO.arIOLinkTx_Place1[2]/InputByte[2] <-> Module 3 (IOL_4/4_I/O-Bytes)/TxPDO/input byte 2
//     MianTask Inputs/G_IO.arIOLinkTx_Place1[2]/InputByte[3] <-> Module 3 (IOL_4/4_I/O-Bytes)/TxPDO/input byte 3
//     MianTask Inputs/G_IO.arIOLinkTx_Place1[3]/InputByte[0] <-> Module 4 (IOL_4/4_I/O-Bytes)/TxPDO/input byte 0
//     MianTask Inputs/G_IO.arIOLinkTx_Place1[3]/InputByte[1] <-> Module 4 (IOL_4/4_I/O-Bytes)/TxPDO/input byte 1
//     MianTask Inputs/G_IO.arIOLinkTx_Place1[3]/InputByte[2] <-> Module 4 (IOL_4/4_I/O-Bytes)/TxPDO/input byte 2
//     MianTask Inputs/G_IO.arIOLinkTx_Place1[3]/InputByte[3] <-> Module 4 (IOL_4/4_I/O-Bytes)/TxPDO/input byte 3
//     MianTask Inputs/G_IO.arIOLinkTx_Place1[4]/InputByte[0] <-> Module 5 (IOL_4/4_I/O-Bytes)/TxPDO/input byte 0
//     MianTask Inputs/G_IO.arIOLinkTx_Place1[4]/InputByte[1] <-> Module 5 (IOL_4/4_I/O-Bytes)/TxPDO/input byte 1
//     MianTask Inputs/G_IO.arIOLinkTx_Place1[4]/InputByte[2] <-> Module 5 (IOL_4/4_I/O-Bytes)/TxPDO/input byte 2
//     MianTask Inputs/G_IO.arIOLinkTx_Place1[4]/InputByte[3] <-> Module 5 (IOL_4/4_I/O-Bytes)/TxPDO/input byte 3
//     MianTask Inputs/G_IO.arIOLinkTx_Place1[5]/InputByte[0] <-> Module 6 (IOL_4/4_I/O-Bytes)/TxPDO/input byte 0
//     MianTask Inputs/G_IO.arIOLinkTx_Place1[5]/InputByte[1] <-> Module 6 (IOL_4/4_I/O-Bytes)/TxPDO/input byte 1
//     MianTask Inputs/G_IO.arIOLinkTx_Place1[5]/InputByte[2] <-> Module 6 (IOL_4/4_I/O-Bytes)/TxPDO/input byte 2
//     MianTask Inputs/G_IO.arIOLinkTx_Place1[5]/InputByte[3] <-> Module 6 (IOL_4/4_I/O-Bytes)/TxPDO/input byte 3
//     MianTask Inputs/G_IO.arIOLinkTx_Place1[6]/InputByte[0] <-> Module 7 (IOL_4/4_I/O-Bytes)/TxPDO/input byte 0
//     MianTask Inputs/G_IO.arIOLinkTx_Place1[6]/InputByte[1] <-> Module 7 (IOL_4/4_I/O-Bytes)/TxPDO/input byte 1
//     MianTask Inputs/G_IO.arIOLinkTx_Place1[6]/InputByte[2] <-> Module 7 (IOL_4/4_I/O-Bytes)/TxPDO/input byte 2
//     MianTask Inputs/G_IO.arIOLinkTx_Place1[6]/InputByte[3] <-> Module 7 (IOL_4/4_I/O-Bytes)/TxPDO/input byte 3
//     MianTask Inputs/G_IO.arIOLinkTx_Place1[7]/InputByte[0] <-> Module 8 (IOL_4/4_I/O-Bytes)/TxPDO/input byte 0
//     MianTask Inputs/G_IO.arIOLinkTx_Place1[7]/InputByte[1] <-> Module 8 (IOL_4/4_I/O-Bytes)/TxPDO/input byte 1
//     MianTask Inputs/G_IO.arIOLinkTx_Place1[7]/InputByte[2] <-> Module 8 (IOL_4/4_I/O-Bytes)/TxPDO/input byte 2
//     MianTask Inputs/G_IO.arIOLinkTx_Place1[7]/InputByte[3] <-> Module 8 (IOL_4/4_I/O-Bytes)/TxPDO/input byte 3
//     MianTask Outputs/G_IO.arIOLinkRx_Place1[0]/OutputByte[0] <-> Module 1 (IOL_4/4_I/O-Bytes)/RxPDO/output byte 0
//     MianTask Outputs/G_IO.arIOLinkRx_Place1[0]/OutputByte[1] <-> Module 1 (IOL_4/4_I/O-Bytes)/RxPDO/output byte 1
//     MianTask Outputs/G_IO.arIOLinkRx_Place1[0]/OutputByte[2] <-> Module 1 (IOL_4/4_I/O-Bytes)/RxPDO/output byte 2
//     MianTask Outputs/G_IO.arIOLinkRx_Place1[0]/OutputByte[3] <-> Module 1 (IOL_4/4_I/O-Bytes)/RxPDO/output byte 3
//     MianTask Outputs/G_IO.arIOLinkRx_Place1[1]/OutputByte[0] <-> Module 2 (IOL_4/4_I/O-Bytes)/RxPDO/output byte 0
//     MianTask Outputs/G_IO.arIOLinkRx_Place1[1]/OutputByte[1] <-> Module 2 (IOL_4/4_I/O-Bytes)/RxPDO/output byte 1
//     MianTask Outputs/G_IO.arIOLinkRx_Place1[1]/OutputByte[2] <-> Module 2 (IOL_4/4_I/O-Bytes)/RxPDO/output byte 2
//     MianTask Outputs/G_IO.arIOLinkRx_Place1[1]/OutputByte[3] <-> Module 2 (IOL_4/4_I/O-Bytes)/RxPDO/output byte 3
//     MianTask Outputs/G_IO.arIOLinkRx_Place1[2]/OutputByte[0] <-> Module 3 (IOL_4/4_I/O-Bytes)/RxPDO/output byte 0
//     MianTask Outputs/G_IO.arIOLinkRx_Place1[2]/OutputByte[1] <-> Module 3 (IOL_4/4_I/O-Bytes)/RxPDO/output byte 1
//     MianTask Outputs/G_IO.arIOLinkRx_Place1[2]/OutputByte[2] <-> Module 3 (IOL_4/4_I/O-Bytes)/RxPDO/output byte 2
//     MianTask Outputs/G_IO.arIOLinkRx_Place1[2]/OutputByte[3] <-> Module 3 (IOL_4/4_I/O-Bytes)/RxPDO/output byte 3
//     MianTask Outputs/G_IO.arIOLinkRx_Place1[3]/OutputByte[0] <-> Module 4 (IOL_4/4_I/O-Bytes)/RxPDO/output byte 0
//     MianTask Outputs/G_IO.arIOLinkRx_Place1[3]/OutputByte[1] <-> Module 4 (IOL_4/4_I/O-Bytes)/RxPDO/output byte 1
//     MianTask Outputs/G_IO.arIOLinkRx_Place1[3]/OutputByte[2] <-> Module 4 (IOL_4/4_I/O-Bytes)/RxPDO/output byte 2
//     MianTask Outputs/G_IO.arIOLinkRx_Place1[3]/OutputByte[3] <-> Module 4 (IOL_4/4_I/O-Bytes)/RxPDO/output byte 3
//     MianTask Outputs/G_IO.arIOLinkRx_Place1[4]/OutputByte[0] <-> Module 5 (IOL_4/4_I/O-Bytes)/RxPDO/output byte 0
//     MianTask Outputs/G_IO.arIOLinkRx_Place1[4]/OutputByte[1] <-> Module 5 (IOL_4/4_I/O-Bytes)/RxPDO/output byte 1
//     MianTask Outputs/G_IO.arIOLinkRx_Place1[4]/OutputByte[2] <-> Module 5 (IOL_4/4_I/O-Bytes)/RxPDO/output byte 2
//     MianTask Outputs/G_IO.arIOLinkRx_Place1[4]/OutputByte[3] <-> Module 5 (IOL_4/4_I/O-Bytes)/RxPDO/output byte 3
//     MianTask Outputs/G_IO.arIOLinkRx_Place1[5]/OutputByte[0] <-> Module 6 (IOL_4/4_I/O-Bytes)/RxPDO/output byte 0
//     MianTask Outputs/G_IO.arIOLinkRx_Place1[5]/OutputByte[1] <-> Module 6 (IOL_4/4_I/O-Bytes)/RxPDO/output byte 1
//     MianTask Outputs/G_IO.arIOLinkRx_Place1[5]/OutputByte[2] <-> Module 6 (IOL_4/4_I/O-Bytes)/RxPDO/output byte 2
//     MianTask Outputs/G_IO.arIOLinkRx_Place1[5]/OutputByte[3] <-> Module 6 (IOL_4/4_I/O-Bytes)/RxPDO/output byte 3
//     MianTask Outputs/G_IO.arIOLinkRx_Place1[6]/OutputByte[0] <-> Module 7 (IOL_4/4_I/O-Bytes)/RxPDO/output byte 0
//     MianTask Outputs/G_IO.arIOLinkRx_Place1[6]/OutputByte[1] <-> Module 7 (IOL_4/4_I/O-Bytes)/RxPDO/output byte 1
//     MianTask Outputs/G_IO.arIOLinkRx_Place1[6]/OutputByte[2] <-> Module 7 (IOL_4/4_I/O-Bytes)/RxPDO/output byte 2
//     MianTask Outputs/G_IO.arIOLinkRx_Place1[6]/OutputByte[3] <-> Module 7 (IOL_4/4_I/O-Bytes)/RxPDO/output byte 3
//     MianTask Outputs/G_IO.arIOLinkRx_Place1[7]/OutputByte[0] <-> Module 8 (IOL_4/4_I/O-Bytes)/RxPDO/output byte 0
//     MianTask Outputs/G_IO.arIOLinkRx_Place1[7]/OutputByte[1] <-> Module 8 (IOL_4/4_I/O-Bytes)/RxPDO/output byte 1
//     MianTask Outputs/G_IO.arIOLinkRx_Place1[7]/OutputByte[2] <-> Module 8 (IOL_4/4_I/O-Bytes)/RxPDO/output byte 2
//     MianTask Outputs/G_IO.arIOLinkRx_Place1[7]/OutputByte[3] <-> Module 8 (IOL_4/4_I/O-Bytes)/RxPDO/output byte 3
//   Rohlik_Expansion/Rohlik_Expansion Instance <-> Place1/Term 27 (EK1100)/DI4
//     MianTask Inputs/G_IO.arDI[4]/Ch[{0..15}] <-> Channel {1..16}/Input  (16 links)
//   Rohlik_Expansion/Rohlik_Expansion Instance <-> Place1/Term 27 (EK1100)/DI5
//     MianTask Inputs/G_IO.arDI[5]/Ch[{0..15}] <-> Channel {1..16}/Input  (16 links)
//   Rohlik_Expansion/Rohlik_Expansion Instance <-> Place1/Term 27 (EK1100)/DO4
//     MianTask Outputs/G_IO.arDO[4]/Ch[{0..15}] <-> Channel {1..16}/Output  (16 links)
//   Rohlik_Expansion/Rohlik_Expansion Instance <-> Place1/Term 27 (EK1100)/DO6
//     MianTask Outputs/G_IO.arDO[6]/Ch[{0..15}] <-> Channel {1..16}/Output  (16 links)
//   Rohlik_Expansion/Rohlik_Expansion Instance <-> Place2
//     MianTask Inputs/G_IO.wcState_place2 <-> Inputs/Frm0WcState
//   Rohlik_Expansion/Rohlik_Expansion Instance <-> Place2/Box 46 (ifm IO-Link Master AL1332)
//     MianTask Inputs/G_IO.arIOLinkQualifier_Place2/CH[{0..7}] <-> TxPDO IO-Link Port Qualifier/Qualifier of IO-Link Ch.{1..8}  (8 links)
//     MianTask Inputs/G_IO.arIOLinkTx_Place2[0]/InputByte[0] <-> Module 1 (IOL_4/4_I/O-Bytes)/TxPDO/input byte 0
//     MianTask Inputs/G_IO.arIOLinkTx_Place2[0]/InputByte[1] <-> Module 1 (IOL_4/4_I/O-Bytes)/TxPDO/input byte 1
//     MianTask Inputs/G_IO.arIOLinkTx_Place2[0]/InputByte[2] <-> Module 1 (IOL_4/4_I/O-Bytes)/TxPDO/input byte 2
//     MianTask Inputs/G_IO.arIOLinkTx_Place2[0]/InputByte[3] <-> Module 1 (IOL_4/4_I/O-Bytes)/TxPDO/input byte 3
//     MianTask Inputs/G_IO.arIOLinkTx_Place2[1]/InputByte[0] <-> Module 2 (IOL_4/4_I/O-Bytes)/TxPDO/input byte 0
//     MianTask Inputs/G_IO.arIOLinkTx_Place2[1]/InputByte[1] <-> Module 2 (IOL_4/4_I/O-Bytes)/TxPDO/input byte 1
//     MianTask Inputs/G_IO.arIOLinkTx_Place2[1]/InputByte[2] <-> Module 2 (IOL_4/4_I/O-Bytes)/TxPDO/input byte 2
//     MianTask Inputs/G_IO.arIOLinkTx_Place2[1]/InputByte[3] <-> Module 2 (IOL_4/4_I/O-Bytes)/TxPDO/input byte 3
//     MianTask Inputs/G_IO.arIOLinkTx_Place2[2]/InputByte[0] <-> Module 3 (IOL_4/4_I/O-Bytes)/TxPDO/input byte 0
//     MianTask Inputs/G_IO.arIOLinkTx_Place2[2]/InputByte[1] <-> Module 3 (IOL_4/4_I/O-Bytes)/TxPDO/input byte 1
//     MianTask Inputs/G_IO.arIOLinkTx_Place2[2]/InputByte[2] <-> Module 3 (IOL_4/4_I/O-Bytes)/TxPDO/input byte 2
//     MianTask Inputs/G_IO.arIOLinkTx_Place2[2]/InputByte[3] <-> Module 3 (IOL_4/4_I/O-Bytes)/TxPDO/input byte 3
//     MianTask Inputs/G_IO.arIOLinkTx_Place2[3]/InputByte[0] <-> Module 4 (IOL_4/4_I/O-Bytes)/TxPDO/input byte 0
//     MianTask Inputs/G_IO.arIOLinkTx_Place2[3]/InputByte[1] <-> Module 4 (IOL_4/4_I/O-Bytes)/TxPDO/input byte 1
//     MianTask Inputs/G_IO.arIOLinkTx_Place2[3]/InputByte[2] <-> Module 4 (IOL_4/4_I/O-Bytes)/TxPDO/input byte 2
//     MianTask Inputs/G_IO.arIOLinkTx_Place2[3]/InputByte[3] <-> Module 4 (IOL_4/4_I/O-Bytes)/TxPDO/input byte 3
//     MianTask Inputs/G_IO.arIOLinkTx_Place2[4]/InputByte[0] <-> Module 5 (IOL_4/4_I/O-Bytes)/TxPDO/input byte 0
//     MianTask Inputs/G_IO.arIOLinkTx_Place2[4]/InputByte[1] <-> Module 5 (IOL_4/4_I/O-Bytes)/TxPDO/input byte 1
//     MianTask Inputs/G_IO.arIOLinkTx_Place2[4]/InputByte[2] <-> Module 5 (IOL_4/4_I/O-Bytes)/TxPDO/input byte 2
//     MianTask Inputs/G_IO.arIOLinkTx_Place2[4]/InputByte[3] <-> Module 5 (IOL_4/4_I/O-Bytes)/TxPDO/input byte 3
//     MianTask Inputs/G_IO.arIOLinkTx_Place2[5]/InputByte[0] <-> Module 6 (IOL_4/4_I/O-Bytes)/TxPDO/input byte 0
//     MianTask Inputs/G_IO.arIOLinkTx_Place2[5]/InputByte[1] <-> Module 6 (IOL_4/4_I/O-Bytes)/TxPDO/input byte 1
//     MianTask Inputs/G_IO.arIOLinkTx_Place2[5]/InputByte[2] <-> Module 6 (IOL_4/4_I/O-Bytes)/TxPDO/input byte 2
//     MianTask Inputs/G_IO.arIOLinkTx_Place2[5]/InputByte[3] <-> Module 6 (IOL_4/4_I/O-Bytes)/TxPDO/input byte 3
//     MianTask Inputs/G_IO.arIOLinkTx_Place2[6]/InputByte[0] <-> Module 7 (IOL_4/4_I/O-Bytes)/TxPDO/input byte 0
//     MianTask Inputs/G_IO.arIOLinkTx_Place2[6]/InputByte[1] <-> Module 7 (IOL_4/4_I/O-Bytes)/TxPDO/input byte 1
//     MianTask Inputs/G_IO.arIOLinkTx_Place2[6]/InputByte[2] <-> Module 7 (IOL_4/4_I/O-Bytes)/TxPDO/input byte 2
//     MianTask Inputs/G_IO.arIOLinkTx_Place2[6]/InputByte[3] <-> Module 7 (IOL_4/4_I/O-Bytes)/TxPDO/input byte 3
//     MianTask Inputs/G_IO.arIOLinkTx_Place2[7]/InputByte[0] <-> Module 8 (IOL_4/4_I/O-Bytes)/TxPDO/input byte 0
//     MianTask Inputs/G_IO.arIOLinkTx_Place2[7]/InputByte[1] <-> Module 8 (IOL_4/4_I/O-Bytes)/TxPDO/input byte 1
//     MianTask Inputs/G_IO.arIOLinkTx_Place2[7]/InputByte[2] <-> Module 8 (IOL_4/4_I/O-Bytes)/TxPDO/input byte 2
//     MianTask Inputs/G_IO.arIOLinkTx_Place2[7]/InputByte[3] <-> Module 8 (IOL_4/4_I/O-Bytes)/TxPDO/input byte 3
//     MianTask Outputs/G_IO.arIOLinkRx_Place2[0]/OutputByte[0] <-> Module 1 (IOL_4/4_I/O-Bytes)/RxPDO/output byte 0
//     MianTask Outputs/G_IO.arIOLinkRx_Place2[0]/OutputByte[1] <-> Module 1 (IOL_4/4_I/O-Bytes)/RxPDO/output byte 1
//     MianTask Outputs/G_IO.arIOLinkRx_Place2[0]/OutputByte[2] <-> Module 1 (IOL_4/4_I/O-Bytes)/RxPDO/output byte 2
//     MianTask Outputs/G_IO.arIOLinkRx_Place2[0]/OutputByte[3] <-> Module 1 (IOL_4/4_I/O-Bytes)/RxPDO/output byte 3
//     MianTask Outputs/G_IO.arIOLinkRx_Place2[1]/OutputByte[0] <-> Module 2 (IOL_4/4_I/O-Bytes)/RxPDO/output byte 0
//     MianTask Outputs/G_IO.arIOLinkRx_Place2[1]/OutputByte[1] <-> Module 2 (IOL_4/4_I/O-Bytes)/RxPDO/output byte 1
//     MianTask Outputs/G_IO.arIOLinkRx_Place2[1]/OutputByte[2] <-> Module 2 (IOL_4/4_I/O-Bytes)/RxPDO/output byte 2
//     MianTask Outputs/G_IO.arIOLinkRx_Place2[1]/OutputByte[3] <-> Module 2 (IOL_4/4_I/O-Bytes)/RxPDO/output byte 3
//     MianTask Outputs/G_IO.arIOLinkRx_Place2[2]/OutputByte[0] <-> Module 3 (IOL_4/4_I/O-Bytes)/RxPDO/output byte 0
//     MianTask Outputs/G_IO.arIOLinkRx_Place2[2]/OutputByte[1] <-> Module 3 (IOL_4/4_I/O-Bytes)/RxPDO/output byte 1
//     MianTask Outputs/G_IO.arIOLinkRx_Place2[2]/OutputByte[2] <-> Module 3 (IOL_4/4_I/O-Bytes)/RxPDO/output byte 2
//     MianTask Outputs/G_IO.arIOLinkRx_Place2[2]/OutputByte[3] <-> Module 3 (IOL_4/4_I/O-Bytes)/RxPDO/output byte 3
//     MianTask Outputs/G_IO.arIOLinkRx_Place2[3]/OutputByte[0] <-> Module 4 (IOL_4/4_I/O-Bytes)/RxPDO/output byte 0
//     MianTask Outputs/G_IO.arIOLinkRx_Place2[3]/OutputByte[1] <-> Module 4 (IOL_4/4_I/O-Bytes)/RxPDO/output byte 1
//     MianTask Outputs/G_IO.arIOLinkRx_Place2[3]/OutputByte[2] <-> Module 4 (IOL_4/4_I/O-Bytes)/RxPDO/output byte 2
//     MianTask Outputs/G_IO.arIOLinkRx_Place2[3]/OutputByte[3] <-> Module 4 (IOL_4/4_I/O-Bytes)/RxPDO/output byte 3
//     MianTask Outputs/G_IO.arIOLinkRx_Place2[4]/OutputByte[0] <-> Module 5 (IOL_4/4_I/O-Bytes)/RxPDO/output byte 0
//     MianTask Outputs/G_IO.arIOLinkRx_Place2[4]/OutputByte[1] <-> Module 5 (IOL_4/4_I/O-Bytes)/RxPDO/output byte 1
//     MianTask Outputs/G_IO.arIOLinkRx_Place2[4]/OutputByte[2] <-> Module 5 (IOL_4/4_I/O-Bytes)/RxPDO/output byte 2
//     MianTask Outputs/G_IO.arIOLinkRx_Place2[4]/OutputByte[3] <-> Module 5 (IOL_4/4_I/O-Bytes)/RxPDO/output byte 3
//     MianTask Outputs/G_IO.arIOLinkRx_Place2[5]/OutputByte[0] <-> Module 6 (IOL_4/4_I/O-Bytes)/RxPDO/output byte 0
//     MianTask Outputs/G_IO.arIOLinkRx_Place2[5]/OutputByte[1] <-> Module 6 (IOL_4/4_I/O-Bytes)/RxPDO/output byte 1
//     MianTask Outputs/G_IO.arIOLinkRx_Place2[5]/OutputByte[2] <-> Module 6 (IOL_4/4_I/O-Bytes)/RxPDO/output byte 2
//     MianTask Outputs/G_IO.arIOLinkRx_Place2[5]/OutputByte[3] <-> Module 6 (IOL_4/4_I/O-Bytes)/RxPDO/output byte 3
//     MianTask Outputs/G_IO.arIOLinkRx_Place2[6]/OutputByte[0] <-> Module 7 (IOL_4/4_I/O-Bytes)/RxPDO/output byte 0
//     MianTask Outputs/G_IO.arIOLinkRx_Place2[6]/OutputByte[1] <-> Module 7 (IOL_4/4_I/O-Bytes)/RxPDO/output byte 1
//     MianTask Outputs/G_IO.arIOLinkRx_Place2[6]/OutputByte[2] <-> Module 7 (IOL_4/4_I/O-Bytes)/RxPDO/output byte 2
//     MianTask Outputs/G_IO.arIOLinkRx_Place2[6]/OutputByte[3] <-> Module 7 (IOL_4/4_I/O-Bytes)/RxPDO/output byte 3
//     MianTask Outputs/G_IO.arIOLinkRx_Place2[7]/OutputByte[0] <-> Module 8 (IOL_4/4_I/O-Bytes)/RxPDO/output byte 0
//     MianTask Outputs/G_IO.arIOLinkRx_Place2[7]/OutputByte[1] <-> Module 8 (IOL_4/4_I/O-Bytes)/RxPDO/output byte 1
//     MianTask Outputs/G_IO.arIOLinkRx_Place2[7]/OutputByte[2] <-> Module 8 (IOL_4/4_I/O-Bytes)/RxPDO/output byte 2
//     MianTask Outputs/G_IO.arIOLinkRx_Place2[7]/OutputByte[3] <-> Module 8 (IOL_4/4_I/O-Bytes)/RxPDO/output byte 3
//   Rohlik_Expansion/Rohlik_Expansion Instance <-> Place2/Term 36 (EK1100)/DI6
//     MianTask Inputs/G_IO.arDI[6]/Ch[{0..15}] <-> Channel {1..16}/Input  (16 links)
//   Rohlik_Expansion/Rohlik_Expansion Instance <-> Place2/Term 36 (EK1100)/DI7
//     MianTask Inputs/G_IO.arDI[7]/Ch[{0..15}] <-> Channel {1..16}/Input  (16 links)
//   Rohlik_Expansion/Rohlik_Expansion Instance <-> Place2/Term 36 (EK1100)/DO5
//     MianTask Outputs/G_IO.arDO[5]/Ch[{0..15}] <-> Channel {1..16}/Output  (16 links)
//   Rohlik_Expansion/Rohlik_Expansion Instance <-> Place2/Term 36 (EK1100)/DO7
//     MianTask Outputs/G_IO.arDO[7]/Ch[{0..15}] <-> Channel {1..16}/Output  (16 links)
//   Rohlik_Expansion/Rohlik_Expansion Instance <-> NC-Task 1 SAF/Axes/autostore1_lift
//     MianTask Inputs/GVL.fb_autoStore1.AxisRef_lift.NcToPlc <-> Outputs/ToPlc
//     MianTask Outputs/GVL.fb_autoStore1.AxisRef_lift.PlcToNc <-> Inputs/FromPlc
//   Rohlik_Expansion/Rohlik_Expansion Instance <-> NC-Task 1 SAF/Axes/autostore1_transfer
//     MianTask Inputs/GVL.fb_autoStore1.AxisRef_transfer.NcToPlc <-> Outputs/ToPlc
//     MianTask Outputs/GVL.fb_autoStore1.AxisRef_transfer.PlcToNc <-> Inputs/FromPlc
//   Rohlik_Expansion/Rohlik_Expansion Instance <-> NC-Task 1 SAF/Axes/autostore2_lift
//     MianTask Inputs/GVL.fb_autoStore2.AxisRef_lift.NcToPlc <-> Outputs/ToPlc
//     MianTask Outputs/GVL.fb_autoStore2.AxisRef_lift.PlcToNc <-> Inputs/FromPlc
//   Rohlik_Expansion/Rohlik_Expansion Instance <-> NC-Task 1 SAF/Axes/autostore2_transfer
//     MianTask Inputs/GVL.fb_autoStore2.AxisRef_transfer.NcToPlc <-> Outputs/ToPlc
//     MianTask Outputs/GVL.fb_autoStore2.AxisRef_transfer.PlcToNc <-> Inputs/FromPlc
//   Rohlik_Expansion/Rohlik_Expansion Instance <-> NC-Task 1 SAF/Axes/lift_motor
//     MianTask Inputs/GVL.fb_loading.AxisRef.NcToPlc <-> Outputs/ToPlc
//     MianTask Inputs/GVL.fb_loading.st_mcAxis.rActTorque <-> Outputs/ToPlc/ActTorque
//     MianTask Outputs/GVL.fb_loading.AxisRef.PlcToNc <-> Inputs/FromPlc
//   Rohlik_Expansion/Rohlik_Expansion Instance <-> NC-Task 1 SAF/Axes/working1_lift_motor
//     MianTask Inputs/GVL.fb_working1.AxisRef_lift.NcToPlc <-> Outputs/ToPlc
//     MianTask Inputs/GVL.fb_working1.st_mcAxis_lift.rActTorque <-> Outputs/ToPlc/ActTorque
//     MianTask Outputs/GVL.fb_working1.AxisRef_lift.PlcToNc <-> Inputs/FromPlc
//   Rohlik_Expansion/Rohlik_Expansion Instance <-> NC-Task 1 SAF/Axes/working1_open_bag
//     MianTask Inputs/GVL.fb_working1.AxisRef_bag.NcToPlc <-> Outputs/ToPlc
//     MianTask Inputs/GVL.fb_working1.st_mcAxis_bag.rActTorque <-> Outputs/ToPlc/ActTorque
//     MianTask Outputs/GVL.fb_working1.AxisRef_bag.PlcToNc <-> Inputs/FromPlc
//   Rohlik_Expansion/Rohlik_Expansion Instance <-> NC-Task 1 SAF/Axes/working2_lift_motor
//     MianTask Inputs/GVL.fb_working2.AxisRef_lift.NcToPlc <-> Outputs/ToPlc
//     MianTask Inputs/GVL.fb_working2.st_mcAxis_lift.rActTorque <-> Outputs/ToPlc/ActTorque
//     MianTask Outputs/GVL.fb_working2.AxisRef_lift.PlcToNc <-> Inputs/FromPlc
//   Rohlik_Expansion/Rohlik_Expansion Instance <-> NC-Task 1 SAF/Axes/working2_open_bag
//     MianTask Inputs/GVL.fb_working2.AxisRef_bag.NcToPlc <-> Outputs/ToPlc
//     MianTask Inputs/GVL.fb_working2.st_mcAxis_bag.rActTorque <-> Outputs/ToPlc/ActTorque
//     MianTask Outputs/GVL.fb_working2.AxisRef_bag.PlcToNc <-> Inputs/FromPlc

CONFIGURATION Rohlik_Expansion
    RESOURCE PLC ON TwinCAT3
        TASK EtherCAT_Task(INTERVAL := T#2ms, PRIORITY := 2);
    END_RESOURCE
END_CONFIGURATION

// ---- 02DUTs/ModuleID.TcDUT
{attribute 'qualified_only'}
{attribute 'strict'}
TYPE ModuleID :
(
	UNKNOWN					:= 0,
	SAFETY					:= 1,
	AIR						:= 2,
	
	
	
	LOADING					:= 3,
	WORKING1				:= 4,
	WORKING2				:= 5,
	
	AUTOSTORE1				:= 6,
	AUTOSTORE2				:= 7,
	
	SAMPLE1					:= 98,
	SAMPLE2					:= 99
);
END_TYPE

// ---- 02DUTs/ST_ChangeIntoProduction.TcDUT
//structure for a visu userwindow, to chnage into productionmode
TYPE ST_ChangeIntoProduction :
STRUCT
	bYes		: BOOL;
	bNo			: BOOL;
	bYesReset	: BOOL;
END_STRUCT
END_TYPE

// ---- Ads/AutostoreControlCommand.TcDUT
{attribute 'qualified_only'}
{attribute 'strict'}
TYPE AutostoreControlCommand :
(
	DO_NOTHING := 0,
	START	:= 1,
	STOP	:= 2
);
END_TYPE

// ---- Ads/DigitalOutputStatus.TcDUT
{attribute 'qualified_only'}
{attribute 'strict'}
TYPE DigitalOutputStatus:
(
        OFF := 0,
        ON := 1
);
END_TYPE

// ---- Ads/EStopStatus.TcDUT
{attribute 'qualified_only'}
{attribute 'strict'}
TYPE EStopStatus:
(
        UNKNOWN := 0, 
		ENGAGED := 1, 
		DISENGAGED := 2
);
END_TYPE

// ---- Ads/E_SAFETYDOOR.TcDUT
{attribute 'qualified_only'}
{attribute 'strict'}
TYPE E_SAFETYDOOR :
(
	IDLE := 0,
	SAFETY,
	LOCKING,
	UNLOCKING,
	UNLOCKED,
	LOCKED,
	WAIT_LOCKED,
	WAIT_UNLOCKED,
	WAIT_UNLOCK_EN,
	REQUEST_LOCK,
	WAIT_ROBOT,
	WATI_LODING_DOOR,
	RESET_SAFETY
);
END_TYPE

// ---- Ads/GeneralStatus.TcDUT
{attribute 'qualified_only'}
{attribute 'strict'}
TYPE GeneralStatus:
( 
	UNKNOWN    := 0,
    READY := 1,
    NOT_READY := 2,
	ERROR := 3
);
END_TYPE

// ---- Ads/InboundToteParams.TcDUT
{attribute 'pack_mode':='1'}
TYPE InboundToteParams :
STRUCT
	source_id : ModelIdentifier; // Identifier for the source inbound line.
	target_id : ModelIdentifier; // Identifier for the target work position.
END_STRUCT
END_TYPE

// ---- Ads/LightCurtainStatus.TcDUT
{attribute 'qualified_only'}
{attribute 'strict'}
TYPE LightCurtainStatus :
(
	UNKNOWN := 0, UNBLOCKED := 1, BLOCKED := 2
);
END_TYPE

// ---- Ads/MachineControlCommand.TcDUT
{attribute 'qualified_only'}
{attribute 'strict'}
TYPE MachineControlCommand :
(
DO_NOTHING := 0,
START := 1, (* Start machine *)
STOP := 2, (* Stop machine *)
RESET := 3 (* Clear machine error status *)
);
END_TYPE

// ---- Ads/MachineControlCommand_1.TcDUT
{attribute 'qualified_only'}
{attribute 'strict'}
TYPE MachineControlCommand_1 :
(
	DO_NOTHING := 0,
	START := 1, (* Start machine *)
	STOP := 2, (* Stop machine *)
	RESET := 3 (* Clear machine error status *)
);
END_TYPE

// ---- Ads/OutboundToteParams.TcDUT
{attribute 'pack_mode':='1'}
TYPE OutboundToteParams :
STRUCT
	source_id : ModelIdentifier; // Identifier for the source inbound line.
	target_id : ModelIdentifier; // Identifier for the target work position.
END_STRUCT
END_TYPE

// ---- Ads/SafetyDoorStatus.TcDUT
{attribute 'qualified_only'}
{attribute 'strict'}
TYPE SafetyDoorStatus:
(
        UNKNOWN := 0, 
		UNLOCKED := 1, 
		LOCKED := 2
);
END_TYPE

// ---- Ads/SensorStatus.TcDUT
{attribute 'qualified_only'}
{attribute 'strict'}
TYPE SensorStatus :
(
	UNKNOWN := 0,
	NO_SIGNAL:=1,
	SIGNAL:=2
);

END_TYPE

// ---- Ads/ST_BagOpen.TcDUT
TYPE ST_BagOpen :
STRUCT
	bag_status				: BagStatus;
	iCnt_sensor_detection	: INT;
	sensor_status			: STRING;
END_STRUCT
END_TYPE

// ---- Ads/UpdateLightTowerParams.TcDUT
{attribute 'pack_mode':='1'}
TYPE UpdateLightTowerParams :
STRUCT
	color 			: UDINT; (* Represents a combination of LightTowerColor values for the colors *)
	flash_period_ms : ULINT; (* Duration in milliseconds for flashing cycle *)
END_STRUCT
END_TYPE

// ---- LogTECH/LogTechStatus.TcDUT
{attribute 'qualified_only'}
{attribute 'strict'}
TYPE LogTechStatus:
(
  	STOPPED			:= 0,
   	RESETTING		:= 1,
   	READY			:= 2,
   	INITIALIZING	:= 3,
 	RUNNING			:= 4,
    STOPPING		:= 5,
   	ERROR			:= 6
);
END_TYPE

// ---- LogTECH/LogTechTransferStatus.TcDUT
{attribute 'qualified_only'}
{attribute 'strict'}
TYPE LogTechTransferStatus:
(
	UNKNOWN					:= 0,
  	READY_TO_RECEIVE		:= 1,
	RECEIVING_TOTE			:= 2,
	RECEIVE_TOTE_FINISHED	:= 3,
	READY_TO_TRANSFER		:= 4,
	TRANSFERING_TOTE		:= 5,//also for stop the process,both stop and error
	TRANSFER_TOTE_FINISHED	:= 6
);
END_TYPE

// ---- Mian/axis/ST_MotionAxis_MC.TcDUT
TYPE ST_MotionAxis_MC :
STRUCT
	rVelocity						: 	LREAL   						;
	rVelocity2						: 	LREAL   						;
	rMaxVelocity					:	LREAL							;	
	rAcceleration					:	LREAL							;
	rMaxAcceleration				:	LREAL							;
	rDeceleration					:	LREAL   						;
	rMaxDeceleration				:	LREAL							;
	rJerk							:	LREAL							;
	rMaxJerk						:	LREAL							;
	rPosition						:	LREAL							;
	rSetPosDistance					:	LREAL							;
	rSetPos							: 	LREAL							;	
	rDistance						:   LREAL							;
	rDistance2						:   LREAL							;	
	
	rActualPosSet					:	LREAL							;//ADD BY EVAN 
	rVelocitySet					: 	LREAL   						;//ADD BY EVAN 	
	xHoming							:	BOOL							;//ADD BY EVAN 
	
	rMaxDistance					:	LREAL							;
	bLimit							:   BOOL							;
	bNegLim							:   BOOL							;
	bPosLim							:	BOOL							;
	bNegSen							:   BOOL							;
	bPosSen							:	BOOL							;
	bPositionSensor					:	BOOL							;
	rHomePos						:	LREAL							;
	rActualPos						:	LREAL							;
	PosDiff							:	LREAL							;
	rActualCurr						:	LREAL							;
	axisDirection					:	MC_Direction					;
	
	rVeloPers						: 	LREAL							;
	rAccPers						: 	LREAL							;   
	rDecPers						: 	LREAL							;                                             					
	SetHomePos						: 	LREAL							;
	HomeVelo						: 	LREAL							;
	PosDiffTarget					: 	LREAL							;
	rFirstpos						: 	LREAL							;
	iAxisID							:	INT								;
	xhsHomingStart					: 	BOOL							;
	xHomingDone						: 	BOOL							;
	xForceControlStart				: 	BOOL							;
	xFoceControlDone				:	BOOL							;	
	xMoveABSDone					: 	BOOL							;
	xMoveRelDone					:	BOOL							;
	bInCouple						:	BOOL							;//Flag Axis is coupled 
    xMuteAxisErrorMessages			:	BOOL							;                                         					
	//Visible/Hide HMI interfaces                   					
	bHomeButtonShow					:	BOOL							; 
	bNegSensorShow					:	BOOL							; 
	bPosSensorShow					:	BOOL							;
	bBacklashShow					:	BOOL							;
	bUnitDegShow					:	BOOL							;
    bJerkShow						:	BOOL							; 
	bStopButtonShow					:	BOOL							; 
	   
	
	bMoveAbsHMI						:	BOOL;
	rVelocityHMI 					: 	LREAL;
	rActualPosHMI					:	LREAL							;//ADD BY EVAN
	bMChomingEnable					:	BOOL							;                                         				
	// backlash compensation                        	
	rBacklashvalue					:	LREAL							;
	xbacklashEnable					:	BOOL							;                        		                					
	bdirFW							:	BOOL							;// on hard stop homing , define the direction of rotation
	
	ModOp					 		: 	SINT							;// Axis operation mode (8 )

//	==============================	Beckhoff Tc2_MC2 library(motion)	==================================
	mcPower 						: 	MC_Power					    ;(*	Axis power, enable/disable																			*)
	mcAxisStates					:	MC_AxisStates					;(*	Driver Feedback, curr motor stage 																	*)
	mcHalt							: 	MC_Halt							;(*	Stops an axis with a defined braking ramp															*)
	mcHome							: 	MC_Home							;(*	Axis homing scenario and execution																	*)
	mcJog							: 	MC_Jog							;(*	Axis Joging BW/FW																					*)	
	mcMoveAbsolute					: 	MC_MoveAbsolute					;(*	Axis GoTo Absolute position																			*)	
	mcMoveRelative					: 	MC_MoveRelative					;(*	Axis GoTo Step by SetPos +/- actual position														*)
	mcMoveVelocity					: 	MC_MoveVelocity					;(*	Axis GoTo with constant velocity														*)
	mcReadStatus					: 	MC_ReadStatus					;(*	Read Axis statuses from driver																		*)
	mcReset							: 	MC_Reset						;(*	Reset Driver																						*)
	mcStop							: 	MC_Stop							;(*	Stop Driver																							*)
	mcReadActualPosition			:	MC_ReadActualPosition			;(*	Read the current axis position																		*)
	mcSetpoint						: 	MC_SetPosition					;(*	Sets the current axis position to a parameterizable value											*)
	mcWriteBoolParameter			: 	MC_WriteBoolParameter			;(*	Write bool param to driver																			*)
	mcReadBoolParameter				:	MC_ReadBoolParameter			;(*	Read bool param from driver																			*)
	mcAxisParameter					:   MC_AxisParameter				;(*	Data type is used in conjunction with function blocks for reading and writing of axis parameters	*)
	CoeWrt							:	FB_EcCoESdoWrite;									
	
//	======================================================================================================	

//
	iSdoWrite	:INT; //6:clear encoder
	sNetID : STRING;
	nSlaveAddr	:UINT;
	nSubIndex	: BYTE;
	nIndex	: WORD;
	
	iCoeWrt	: INT;
	rToqueLimitSet	: LREAL	:= 350;
	rToqueSet	: LREAL;
	rActTorque	AT%I*	: LREAL ;
	xTorqueErr	: BOOL;
	bTouchTorque		: BOOL;
	bTouque_control_enable	: BOOL;
	iAxis	: WORD;
	// digitalInputs     AT%I*  : UDINT;//bit16:limit_positive;bit17:limit_negative;bit18:limit_home//inovance
	limit_sensor_positive:BOOL;
    limit_sensor_negative:BOOL;
    limit_sensor_home:BOOL;

END_STRUCT
END_TYPE

// ---- Mian/DUTs/Buffer_roller.TcDUT
TYPE Buffer_roller :
STRUCT
	roller			: ARRAY[0..1] OF Roller;
	photo_sensor	: ARRAY[0..1] OF BOOL;
	mcAxis			: FB_MotionAxis_MC;
	st_mcAxis 		: ST_MotionAxis_MC;
	AxisRef			: AXIS_REF;
END_STRUCT
END_TYPE

// ---- Mian/DUTs/E_Condition.TcDUT
{attribute 'qualified_only'}
{attribute 'strict'}
TYPE E_Condition :
(
	IDLE 				:= 0,
	PLACE_MOUDULE_UP	:= 1,
	PLACE_MOUDULE_DOWN	:= 2,
	BAG_OPENED			:= 3,
	BAG_CLOSED			:= 4,
	NO_TOTE				:= 5,
	TOTE_IN				:= 6,
	READY_LOADING_TOTE	:= 7,
	TOTE_READY			:= 8
	
);
END_TYPE

// ---- Mian/DUTs/E_LoadingStates.TcDUT

{attribute 'qualified_only'}
{attribute 'strict'}
TYPE E_LoadingStates :
(
	IDLE := 0,
	INIT,
	CHECK,
	WAIT,
	WAIT_1,
	DETECTION,
	LOADING,
	UNLOADING,
	WAIT_WORKING1_READY_LOAD,
	WAIT_WORKING2_READY_LOAD,
	LIFT_POSITION_LOAD,
	LIFT_POSITION_UNLOAD,
	LIFT_UP,
	ROLLER_LOAD,
	ROLLER_UNLOAD_WORKING1,
	ROLLER_UNLOAD_WORKING2,
	WAIT_FINISH_OUTBOUND1,
	WAIT_FINISH_OUTBOUND2,
	AGING_STATE_0,
	AGING_STATE_1,
	DONE,
	WAIT_READY_TO_TRANSFER,
	LOAD_UP_POSITION,
	LOAD_DOWN_POSITION,
	ROLLER_Y_LOAD,
	WORKING1_INBOUND_TOTE,
	WORKING2_INBOUND_TOTE,
	ERROR
);
END_TYPE

// ---- Mian/DUTs/E_SampleStates.TcDUT
{attribute 'qualified_only'}
{attribute 'strict'}
TYPE E_SampleStates :
(
	IDLE := 0,
	INIT,
	CHECK,
	WAIT,
	WAIT_ON,
	WAIT_OFF,
	DETECTION,
	LAMP_ON,
	LAMP_OFF,
	DONE,

	ERROR
);
END_TYPE

// ---- Mian/DUTs/E_AutoStore_States.TcDUT
{attribute 'qualified_only'}
{attribute 'strict'}
TYPE E_AutoStore_States :
(
	IDLE := 0,
	INIT,
	CHECK,//IF AT WORKING POSITION 
	WAIT,
	WAIT_CMD,
	STATUS_DETECTED,
	START,
	STOP,
	LIFT_MOVE_DOWN,
	LIFT_DOWN_SENSOR_DETECTED,
	TRANSFER_MOVE_WORKING,
	TRANSFER_MOVE_FEEDING,
	TRANSFER_WORKING_SENSOR_DETECTED,
	TRANSFER_FEEDING_SENSOR_DETECTED,
	LIFT_MOVE_UP,
	DONE,

	ERROR
);
END_TYPE

// ---- Mian/DUTs/Inbound.TcDUT
TYPE Inbound :
STRUCT
	roller	: Roller;
	//photo_sensor_mute	 : FB_DigitalInput;
	//photo_sensor	: FB_DigitalInput;
	photo_sensor:ARRAY[0..1]OF FB_DigitalInput;
END_STRUCT
END_TYPE

// ---- Mian/DUTs/Outbound.TcDUT
TYPE Outbound :
STRUCT
	roller	: Roller;
	photo_sensor	: FB_DigitalInput;
END_STRUCT
END_TYPE

// ---- Mian/DUTs/Roller_y.TcDUT
TYPE Roller_y :
STRUCT
	roller	: Roller;
	photo_sensor	: ARRAY[0..1] OF FB_DigitalInput;
END_STRUCT
END_TYPE

// ---- Mian/DUTs/ServerityLevelType.TcDUT
{attribute 'qualified_only'}
{attribute 'strict'}
TYPE ServerityLevelType :
(
	SERVICE := 0,
	ERROR,
	WARNING,
	INFO,
	DEBUG
);
END_TYPE

// ---- Mian/DUTs/ST_control_pannel.TcDUT
TYPE ST_control_pannel :
STRUCT
	button_start		: BOOL;
	button_stop			: BOOL;
	button_reset		: BOOL;
	button_power		: BOOL;
	
	lamp_start			: BOOL;
	lamp_stop			: BOOL;
	lamp_reset			: BOOL;
	
END_STRUCT
END_TYPE

// ---- Mian/DUTs/ToteSubsystemWorkflowStatus.TcDUT
{attribute 'qualified_only'}
{attribute 'strict'}
TYPE ToteSubsystemWorkflowStatus:
(
	UNKNOWN					:=0,
  	IDLE					:=1,
	INITIALIZING			:=2,
 	WAITING_FOR_NEW_TOTE	:=3,
 	INBOUNDING				:=4,
  	BAG_OPENING				:=5,
   	WAITING_FOR_UNLOADING	:=6,
  	OUTBOUNDING				:=7
	
);
END_TYPE

// ---- PubSub/E_Topics.TcDUT
TYPE E_Topics :
(
	UNKNOWN 							:= 0, 
	WORKING1_INBOUND_TOTE				:= 1, //publish from inbound_tote_request	
	WORKING1_OUTBOUND_TOTE				:= 2, //publish from outbound_tote_request
	LOADING_BEGIN_OUTBOUND_WOKING1		:= 3, 
	LOADING_END_OUTBOUND_WOKING1		:= 4,
	WORKING1_BEGIN_INBOUND				:= 5,
	WORKING1_ABORT_INBOUND				:= 6,
	WORKING1_ABORT_OUTBOUND				:= 7,
	WORKING2_INBOUND_TOTE				:= 8, //publish from inbound_tote_request
	WORKING2_OUTBOUND_TOTE				:= 9, //publish from outbound_tote_request
	LOADING_BEGIN_OUTBOUND_WOKING2		:= 10,
	LOADING_END_OUTBOUND_WOKING2		:= 11,
	WORKING2_BEGIN_INBOUND				:= 12,
	WORKING2_ABORT_INBOUND				:= 13,
	WORKING2_ABORT_OUTBOUND				:= 14,
	RESET_WAITING_FOR_NEW_SPACE			:= 15,//publish from loding module while wait new tote from logtech too long
	AUTOSTORE1_EXCHANGE					:= 16,
	AUTOSTORE2_EXCHANGE					:= 16,
	SAMPLE_SUBSCRRIBE_1,
	SAMPLE_SUBSCRRIBE_2,
	SAMPLE_SUBSCRRIBE_3,
	NUMBER_OF_TOPICS
);
END_TYPE

// ---- PubSub/KeyAndValue.TcDUT
TYPE KeyAndValue :
STRUCT
	Key : STRING;
	Value : string;
END_STRUCT
END_TYPE

// ---- PubSub/SubscriberCell.TcDUT
TYPE SubscriberCell :
STRUCT
	occupied	: BOOL;
	sTopic	   	: STRING;
	sInstance	: STRING;
	subscriber 	: I_SubCallback;
END_STRUCT
END_TYPE

// ---- GVLs/GVL.TcGVL
{attribute 'qualified_only'}
VAR_GLOBAL

//	fb_mcp						: FB_mcp;   //  1# Robot+Lighttower+Safetydoor  IO-Mapping
//	fb_mcp_2    				: FB_mcp_1; //  2# Robot+Lighttower+Safetydoor  IO-Mapping
	
	fb_mcp_1						: FB_mcp;//  1# Robot+Lighttower+Safetydoor  IO-Mapping
	fb_mcp_2						: FB_mcp;//  1# Robot+Lighttower+Safetydoor  IO-Mapping
	
	status						: MachineStatus := MachineStatus.STOPPED;
	
	iAng_airPress_left		AT%I*	:INT;
	iAng_airPress_right      AT%I*	:INT;
	aiFlow 				AT%I*	:INT;
	
	iAng_AirFlow_left 		AT%I*	:INT;
	iAng_AirFlow_right 		AT%I*	:INT;


	PackTags					: ST_PackMLv30;					//PackTags
	PackTags1					: ST_PackMLv30;					//PackTags
	PackTags2					: ST_PackMLv30;					//PackTags

	nVisuProductCommand			: DINT;							//Products to produce
	
	nVisuProductCommand_2		: DINT;							//Products to produce

	bButtonProductionReq		: BOOL;							//TRUE when a mode change to PRODUCTION is requested
	bButtonProductionReq_2		: BOOL;							//TRUE when a mode change to PRODUCTION is requested
	stChangeIntoProduction		: ST_ChangeIntoProduction;		//Result of command box "Change to Production requested"

	aUnitInfo					: ARRAY [1..12] OF ST_UnitInfo;	//Array includes the states and modes of machineunits	
	aCaption					: ARRAY [1..12] OF STRING := ['F1','F2','F3','F4','F5','F6','F7','F8','F9','F10','F11','F12'];
	aKeyPressed					: ARRAY [1..12] OF BOOL;	

	aUnitInfo_2					: ARRAY [1..12] OF ST_UnitInfo;	//Array includes the states and modes of machineunits	
	aCaption_2					: ARRAY [1..12] OF STRING := ['F1','F2','F3','F4','F5','F6','F7','F8','F9','F10','F11','F12'];
	aKeyPressed_2				: ARRAY [1..12] OF BOOL;		
	
	alarm						: ST_Alarm;
	alarm_empty					: ST_Alarm;
	alarm_temp_loading			: ST_Alarm;
	alarm_temp_working1			: ST_Alarm;
	alarm_temp_working2			: ST_Alarm;
	fbWriteLog					: FB_WriteLog;
	bWrite						: BOOL;
	str							: STRING;
	
	alarms_hmi		: ARRAY[1..20] OF ST_Alarm_Hmi;
	alarms1_hmi		: ARRAY[1..20] OF ST_Alarm_Hmi;
	alarms2_hmi		: ARRAY[1..20] OF ST_Alarm_Hmi;
	
	pml_adminAlarm				: PML_AdminAlarm;	
	

	
	

	fb_sample					: FB_Sample;
	fb_loading					: FB_loading_tote;
	fb_working1					: FB_working_tote;
	fb_working2					: FB_working_tote;
	fb_autoStore1				: FB_autoStore;
	fb_autoStore2				: FB_autoStore;
	
	PubSubService				: PubSubService;
	
	bRightSensor_Shild			: BOOL;
	bLeftSensor_Shild			: BOOL;
	

	//----------------------------------------tryrun ----------------------------
//	iLeftSizeToteLoaded			: INT;
//	iRightSizeToteLoaded		: INT;
//	bTryRunMode					: BOOL;
//	bTryRunStart				: BOOL;
//	bTryRunFrequency			: BOOL;
//	tTryRun						: TON;
//	tTryRunLeft1				: TON;
//	tTryRunLeft2				: TON;
//	tTryRunRight1				: TON;
//	tTryRunRight2				: TON;
	
	
	
END_VAR

VAR_GLOBAL CONSTANT
	iAlarm_max					: INT:= 20;
	MAX_PUB_SUB_DATA			: INT:=	19;
END_VAR

// ---- GVLs/G_HMI.TcGVL
{attribute 'qualified_only'}
VAR_GLOBAL
	iMainFrame 		: INT;
	iPML_mainFrame	: INT;

	bInit			: BOOL;
	bAging_test		: BOOL	:= FALSE;
	
	sLoginnedUser	: STRING;
	bDisplay:BOOL;
	xLift_Load : BOOL;
	xWorking1_Load : BOOL;
	xWorking1_Unload : BOOL;
	xWorking2_Load : BOOL;
	xWorking2_Unload : BOOL;
	
	
	bLeftDoorUnlock_Request_HMI 	:  BOOL;	//FALSE means lock 	 
	bRightDoorUnlock_Request_HMI 	:  BOOL;	//FALSE means lock 	
END_VAR

// ---- GVLs/G_IO.TcGVL
{attribute 'global_init_slot' := '40600'}
VAR_GLOBAL CONSTANT
	{attribute 'global_init_slot'}
	DiMouduleMAX 			:	INT	:=	30;
	{attribute 'global_init_slot'}
	DOMODULEMAX 			:	INT	:=	30;
	{attribute 'global_init_slot'}
	SiMouduleMAX 			:	INT	:=	16;
	{attribute 'global_init_slot'}
	SoMODULEMAX 			:	INT	:=	16;	
END_VAR

VAR_GLOBAL
	arDI	AT%I*		: ARRAY[0..DiMouduleMAX ] OF ST_IO_16;		//  links to Digital input  Modules 
	arDO	AT%Q*		: ARRAY[0..DOMODULEMAX ] OF ST_IO_16;		//  links to Digital output Modules	
	arSI	AT%I*		: ARRAY[0..SiMouduleMAX ] OF ST_SafetyIO;	//  links to safety input  Modules
	arSO	AT%Q*		: ARRAY[0..SOMODULEMAX ] OF ST_SafetyIO;	//  links to safety output  Modules
	
	
	arIOLinkTx_Lift  AT%I*			: ARRAY[0..7 ] OF ST_Ifm_TX;
	arIOLinkTx_Place1  AT%I*		: ARRAY[0..7 ] OF ST_Ifm_TX;
	arIOLinkTx_Place2  AT%I*		: ARRAY[0..7 ] OF ST_Ifm_TX;
	
	arIOLinkRx_Lift  AT%Q*			: ARRAY[0..7 ] OF ST_Ifm_RX;
	arIOLinkRx_Place1  AT%Q*		: ARRAY[0..7 ] OF ST_Ifm_RX;
	arIOLinkRx_Place2  AT%Q*		: ARRAY[0..7 ] OF ST_Ifm_RX;
	
	arIOLinkQualifier_Lift  AT%I*	: ST_Ifm_Qualifier ;
	arIOLinkQualifier_Place1  AT%I*	: ST_Ifm_Qualifier ;
	arIOLinkQualifier_Place2  AT%I*	: ST_Ifm_Qualifier ;
/////////////////////////ETHERCAT BUS STATE/////////////////////
	wcState_mcp			AT%I*	: UINT;
	wcState_lift		AT%I*	: UINT;
	wcState_place1		AT%I*	: UINT;
	wcState_place2		AT%I*	: UINT;
	devState_Device1	AT%I*	: UINT;
END_VAR

// ---- Mian/FB_working_tote.TcPOU
FUNCTION_BLOCK FB_working_tote EXTENDS FB_Generic
VAR_IN_OUT
	
END_VAR
VAR_INPUT

	
END_VAR
VAR_OUTPUT
	error_status	: OrderToteErrorStatus := OrderToteErrorStatus.UNKNOWN;	
	
	bag_opening_status	:ARRAY[0..1]OF BagOpeningStatus;
END_VAR
VAR
	eStates				: E_WorkingStates	:= E_WorkingStates.IDLE;
	eStateTemp			: E_WorkingStates	:= E_WorkingStates.IDLE;
	tote_status			: ToteStatus;
	outboundTote_status	: ToteStatus;
	

//	bag_opening_status_0	: REFERENCE TO BagOpeningStatus;
//	bag_opening_status_1	: REFERENCE TO BagOpeningStatus;
	bagOpen_Status			: ARRAY[0..1] OF ST_BagOpen;
	bagOpenInit_Status		: ARRAY[0..1] OF ST_BagOpen;
	
	iCount_sensor_detection	: ARRAY [0..1] OF INT;
	strLog_bagopen_detection	: STRING;
	
//	bOpen_bag_detection		: BOOL	:= TRUE;
//	bOpen_bag_detection_0	: BOOL	:= TRUE;
//	bOpen_bag_detection_1	: BOOL	:= TRUE;
	
	logtech_control_command	: LogTechControlCmd;
	logtech_status	:LogTechStatus;
	logtech_transfer_status	: LogTechTransferStatus;
	//rPos_bag_closed_step_0	: REAL;  //半开袋位置设定
	bRobot_in_safety_place	: BOOL:=TRUE;
///////

	valve_lift			: Valve;
	roller_inbound		: Inbound;
	roller_outbound		: Outbound;
	roller_outbound_assist	: Outbound;
	photo_sensor_tote_detection: FB_DigitalInput;
	
    BagOpening_Detection	: ARRAY[0..7] OF BOOL;
	sensor_cover			: ARRAY[0..1] OF BOOL;
	EDM_KM			    : BOOL;
	
	mcAxis_lift 		: FB_MotionAxis_MC;
	st_mcAxis_lift 		: ST_MotionAxis_MC;
	AxisRef_lift		: AXIS_REF;
	
	mcAxis_bag 			: FB_MotionAxis_MC;
	st_mcAxis_bag		: ST_MotionAxis_MC;
	AxisRef_bag			: AXIS_REF;		
	
//	xLoading : BOOL;
//	xUnloading : BOOL;
	xInbound	: BOOL;
	xOutbound	: BOOL;
	rPos_bag_closed_step_0	: REAL;
	
	
	xBeginInbound	: BOOL;
	xAbortInbound	: BOOL;
	xAbortOutbound	: BOOL;
	
	rTrig1	: R_TRIG;
	fTrig1	: F_TRIG;
	str4debug	: STRING;
	eState_temp1	: STRING;
	state_track		: STRING(255);
	
	
	
	stSubModuleInfo		: ARRAY [1..iSubModule] OF ST_PMLSubUnitInfo;	//Informations about the Subunits
	bMachineStartedUp	: BOOL;
END_VAR

VAR CONSTANT
	rMax_lift	: REAL	:= 135;
	rMin_lift	: REAL	:= -0.5;
	rMax_bag	: REAL	:= 56;
	rMin_bag	: REAL	:= -0.5;	
	
	iSubModule		: UDINT:=1;
END_VAR

VAR PERSISTENT
	rPos_lift_up				: REAL;
	rPos_lift_down				: REAL;
	rPos_bag_opened				: REAL;
	rPos_bag_closed				: REAL;	
	rPos_bag_preopen			: REAL;
	iDelay_sensor_detection		: INT;
	iSensor_detection_setting	: ARRAY [0..1] OF INT;
	bUsingOpenBag				: BOOL;
END_VAR

SUPER^();
infoLevel	:= ServerityLevelType.WARNING;
IF sInstanceName='working1' THEN
	IF NOT subscribed THEN
		GVL.PubSubService.Subscribe(E_Topics.WORKING1_INBOUND_TOTE,sInstanceName,THIS^);
		GVL.PubSubService.Subscribe(E_Topics.WORKING1_OUTBOUND_TOTE,sInstanceName,THIS^);
		GVL.PubSubService.Subscribe(E_Topics.WORKING1_BEGIN_INBOUND,sInstanceName,THIS^);
		GVL.PubSubService.Subscribe(E_Topics.WORKING1_ABORT_INBOUND,sInstanceName,THIS^);
		GVL.PubSubService.Subscribe(E_Topics.WORKING1_ABORT_OUTBOUND,sInstanceName,THIS^);
		subscribed	:= TRUE;
	END_IF
END_IF
IF sInstanceName='working2' THEN
	IF NOT subscribed THEN
		GVL.PubSubService.Subscribe(E_Topics.WORKING2_INBOUND_TOTE,sInstanceName,THIS^);
		GVL.PubSubService.Subscribe(E_Topics.WORKING2_OUTBOUND_TOTE,sInstanceName,THIS^);	
		GVL.PubSubService.Subscribe(E_Topics.WORKING2_BEGIN_INBOUND,sInstanceName,THIS^);
		GVL.PubSubService.Subscribe(E_Topics.WORKING2_ABORT_INBOUND,sInstanceName,THIS^);
		GVL.PubSubService.Subscribe(E_Topics.WORKING2_ABORT_OUTBOUND,sInstanceName,THIS^);

		subscribed	:= TRUE;
	END_IF
END_IF


//bag_opening_status_0	REF= MAIN.tote_1.working1_tote.bag_opening_status_0;
//bag_opening_status_1	REF= MAIN.tote_1.working2_tote.bag_opening_status_1;

bagOpenInit_Status[0].bag_status				:=BagStatus.UNOPENED;
bagOpenInit_Status[0].iCnt_sensor_detection		:=0;
bagOpenInit_Status[0].sensor_status				:='';
bagOpenInit_Status[1].bag_status				:=BagStatus.UNOPENED;
bagOpenInit_Status[1].iCnt_sensor_detection		:=0;
bagOpenInit_Status[1].sensor_status				:='';
////////////////////////////////////////////////mechanical error///////////////////////////////////////////////////
IF GVL.fb_loading.tote_status=ToteStatus.MECHANICAL_ERROR THEN
	tote_status	:= ToteStatus.MECHANICAL_ERROR;
END_IF
////////////////////////////////////////////////electrical error///////////////////////////////////////////////////
rTrig_electricalError[1](CLK:= st_mcAxis_lift.mcReadStatus.Error);
rTrig_electricalError[2](CLK:= st_mcAxis_bag.mcReadStatus.Error);
rTrig_electricalError[3](CLK:= roller_inbound.roller.err.Q);
rTrig_electricalError[4](CLK:= roller_outbound.roller.err.Q);
rTrig_electricalError[5](CLK:= roller_outbound_assist.roller.err.Q);
IF sInstanceName='working1' THEN
	IF GVL.PackTags1.Status.StateCurrent<>E_PMLState.ePMLState_Resetting THEN
		FOR i:=1 TO 10 DO
			IF rTrig_electricalError[i].Q THEN
				THIS^.packTags.Admin.Alarm[i].ID	:= i;
				CASE i OF
					1:
						THIS^.packTags.Admin.Alarm[1].Message	:= GenerateErrorMsg(errorType:='E',iState := i,errorMsg:='lift axis is in error state.');
					2:
						THIS^.packTags.Admin.Alarm[2].Message	:= GenerateErrorMsg(errorType:='E',iState := i,errorMsg:='open bag axis of working is in error state.');
					3:
						THIS^.packTags.Admin.Alarm[3].Message	:= GenerateErrorMsg(errorType:='E',iState := i,errorMsg:='inbound roller is in error state.');
					4:
						THIS^.packTags.Admin.Alarm[4].Message	:= GenerateErrorMsg(errorType:='E',iState := i,errorMsg:='outbound roller is in error state.');
					5:
						THIS^.packTags.Admin.Alarm[5].Message	:= GenerateErrorMsg(errorType:='E',iState := i,errorMsg:='outbound assist roller is in error state.');
				END_CASE
					tote_status	:= ToteStatus.ELECTRICAL_ERROR;
					GVL.pml_adminAlarm.M_SetAlarm(stAdmin:=GVL.PackTags1.Admin,stAlarm := THIS^.packTags.Admin.Alarm[i]);			
			END_IF
		END_FOR
	END_IF	
END_IF
IF sInstanceName='working2' THEN
	IF GVL.PackTags2.Status.StateCurrent<>E_PMLState.ePMLState_Resetting THEN
		FOR i:=1 TO 10 DO
			IF rTrig_electricalError[i].Q THEN
				THIS^.packTags.Admin.Alarm[i].ID	:= i;
				CASE i OF
					1:
						THIS^.packTags.Admin.Alarm[1].Message	:= GenerateErrorMsg(errorType:='E',iState := i,errorMsg:='lift axis is in error state.');
					2:
						THIS^.packTags.Admin.Alarm[2].Message	:= GenerateErrorMsg(errorType:='E',iState := i,errorMsg:='open bag axis of working is in error state.');
					3:
						THIS^.packTags.Admin.Alarm[3].Message	:= GenerateErrorMsg(errorType:='E',iState := i,errorMsg:='inbound roller is in error state.');
					4:
						THIS^.packTags.Admin.Alarm[4].Message	:= GenerateErrorMsg(errorType:='E',iState := i,errorMsg:='outbound roller is in error state.');
					5:
						THIS^.packTags.Admin.Alarm[5].Message	:= GenerateErrorMsg(errorType:='E',iState := i,errorMsg:='outbound assist roller is in error state.');
				END_CASE	
				GVL.pml_adminAlarm.M_SetAlarm(stAdmin:=GVL.PackTags2.Admin,stAlarm := THIS^.packTags.Admin.Alarm[i]);			
			END_IF
		END_FOR
	END_IF	
END_IF


//rTrig1(CLK:=xInbound);
//IF rTrig1.Q THEN
//	eState_temp1	:= '';
//	str4debug:='';
//	str4debug	:= CONCAT(STR1:=sInstanceName,STR2:='-');
//	str4debug	:= CONCAT(STR1:=str4debug,STR2:=DINT_TO_STRING(eState));
//	str4debug	:= CONCAT(STR1:=str4debug,STR2:='-');
//	str4debug	:= CONCAT(STR1:=str4debug,STR2:=strState);
//	str4debug	:= CONCAT(STR1:=str4debug,STR2:='-');
//	str4debug	:= CONCAT(STR1:=str4debug,STR2:='inbound');
//	str4debug	:= CONCAT(STR1:=str4debug,STR2:='-');
//	str4debug	:= CONCAT(STR1:=str4debug,STR2:='ON');
//	ADSLOGSTR(msgCtrlMask:=ADSLOG_MSGTYPE_LOG,msgFmtStr:=str4debug,strArg:='');
//END_IF
//fTrig1(CLK:=xInbound);
//IF eState_temp1<>strState THEN
//	eState_temp1	:= strState;
//	state_track	:= CONCAT(STR1:=state_track,STR2:=eState_temp1);
//	state_track	:= CONCAT(STR1:=state_track,STR2:='->');
//END_IF
//IF fTrig1.Q THEN
//	str4debug:='';
//	str4debug	:= CONCAT(STR1:=sInstanceName,STR2:='-');
//	str4debug	:= CONCAT(STR1:=str4debug,STR2:=DINT_TO_STRING(eState));
//	str4debug	:= CONCAT(STR1:=str4debug,STR2:='-');
//	str4debug	:= CONCAT(STR1:=str4debug,STR2:=state_track);
//	str4debug	:= CONCAT(STR1:=str4debug,STR2:='-');
//	str4debug	:= CONCAT(STR1:=str4debug,STR2:='inbound');
//	str4debug	:= CONCAT(STR1:=str4debug,STR2:='-');	
//	str4debug	:= CONCAT(STR1:=str4debug,STR2:='OFF');
//	ADSLOGSTR(msgCtrlMask:=ADSLOG_MSGTYPE_LOG,msgFmtStr:=str4debug,strArg:='');
//END_IF
IF sInstanceName='working1' THEN
	GVL.fb_autoStore1(	eModeCommand:=eModeCommand,
						eCommand:=eCommand,
						eMode	=>,
						eState =>stSubModuleInfo[1].eState
					);
	stSubModuleInfo[1].Active			:= TRUE;
	IF  GVL.fb_autoStore1.bUndefinedDone THEN
		bUndefinedDone := TRUE;
	END_IF	
END_IF
IF sInstanceName='working2' THEN
	GVL.fb_autoStore2(	eModeCommand:=eModeCommand,
						eCommand:=eCommand,
						eMode	=>,
						eState =>stSubModuleInfo[1].eState
					);
	stSubModuleInfo[1].Active			:= TRUE;
	IF  GVL.fb_autoStore2.bUndefinedDone THEN
		bUndefinedDone := TRUE;
	END_IF		
END_IF


IF bUndefinedDone AND NOT bMachineStartedUp THEN
	eCommand	:= ePMLCommand_Abort;
	bMachineStartedUp			:= TRUE;
END_IF
//The fbStateMachine from FB_Machine gets the Information about the states and activity from the subunits
fbStateMachine.stSubUnitInfoRef.ArraySize		:= SIZEOF(stSubModuleInfo);
fbStateMachine.stSubUnitInfoRef.NoOfSubUnits	:= iSubModule;
fbStateMachine.stSubUnitInfoRef.pArray			:= ADR(stSubModuleInfo);

(*
Description: 
the callback that will be invoked when there is a publish for what the subscriber was subscribed to.
*)
METHOD Callback
VAR_INPUT
	data : PubSubData;
END_VAR

IF sInstanceName='working1' THEN
	CASE data.Topic OF	
		E_Topics.WORKING1_INBOUND_TOTE:
			IF NOT xInbound AND NOT xOutbound THEN
				xInbound	:= TRUE;
			END_IF
		E_Topics.WORKING1_OUTBOUND_TOTE:
			IF NOT xInbound AND NOT xOutbound THEN
				xOutbound	:= TRUE;
			END_IF
		E_Topics.WORKING1_BEGIN_INBOUND:
			xBeginInbound	:= TRUE;	
		E_Topics.WORKING1_ABORT_INBOUND:
			IF eStates=E_WorkingStates.WAIT_NEW_TOTE THEN
				subData.Topic	:= E_Topics.LOADING_END_OUTBOUND_WOKING1;
				GVL.PubSubService.Publish(topic:=E_Topics.LOADING_END_OUTBOUND_WOKING1,data:= subData);		
				xAbortInbound	:= TRUE;
			END_IF	
		E_Topics.WORKING1_ABORT_OUTBOUND:
			xAbortOutbound	:= TRUE;			

	END_CASE
END_IF
IF sInstanceName='working2' THEN
	CASE data.Topic OF	
		E_Topics.WORKING2_INBOUND_TOTE:
			IF NOT xInbound AND NOT xOutbound THEN
				xInbound	:= TRUE;
			END_IF
		E_Topics.WORKING2_OUTBOUND_TOTE:
			IF NOT xInbound AND NOT xOutbound THEN
				xOutbound	:= TRUE;
			END_IF
		E_Topics.WORKING2_BEGIN_INBOUND:
			xBeginInbound	:= TRUE;	
		E_Topics.WORKING2_ABORT_INBOUND:
			IF eStates=E_WorkingStates.WAIT_NEW_TOTE THEN
				subData.Topic	:= E_Topics.LOADING_END_OUTBOUND_WOKING2;
				GVL.PubSubService.Publish(topic:=E_Topics.LOADING_END_OUTBOUND_WOKING2,data:= subData);				
				xAbortInbound	:= TRUE;
			END_IF
		E_Topics.WORKING2_ABORT_OUTBOUND:
			xAbortOutbound	:= TRUE;	
		
	END_CASE
END_IF
END_METHOD

{attribute 'object_name' := 'M_Aborting'}
METHOD M_Aborting
CASE fbUnitModeManager.eModeStatus OF	
	ePMLProtUnitMode_Production, ePMLProtUnitMode_Manual:		
		roller_inbound.roller.forward	:= FALSE;
		roller_outbound.roller.forward		:= FALSE;
		roller_outbound_assist.roller.forward	:= FALSE;	
		st_mcAxis_lift.mcMoveAbsolute.Execute	:= FALSE;
		st_mcAxis_bag.mcMoveAbsolute.Execute	:= FALSE;
		st_mcAxis_lift.mcStop.Execute			:= TRUE;
		st_mcAxis_bag.mcStop.Execute			:= TRUE;	
		xInbound	:= FALSE;
		xOutbound	:= FALSE;
		iAging_test	:= 0;
		CASE tote_status OF
			ToteStatus.AWAITING_INBOUND_AVAILABILITY:
			//
			ToteStatus.AWAITING_OUTBOUND_AVAILABILITY:
			//
			ToteStatus.BAG_OPEN_FAILED:
			//
			ToteStatus.DOWNSTREAM_NOT_READY:
			//
			ToteStatus.ELECTRICAL_ERROR:
			//
			ToteStatus.INBOUNDING:
			//
			ToteStatus.LOADED:
			//
			ToteStatus.MECHANICAL_ERROR:
			//
			ToteStatus.OUTBOUNDING:
			//
			ToteStatus.PERTURBING:
			//
		END_CASE
		M_StateComplete();
			
	ePMLProtUnitMode_Maintenance, ePMLUnitMode_Service:
		
		M_StateComplete();
END_CASE
END_METHOD

METHOD M_agingTest : BOOL
VAR_INPUT
	rVelocity_percent	: REAL;
END_VAR
ton_aging_test();
CASE iAging_test OF
	0://
	
	1://run forward
		ton_aging_test.PT	:= T#5S;
		ton_aging_test.IN	:= TRUE;
		st_mcAxis_lift.mcMoveAbsolute.Execute	:= TRUE;						
		st_mcAxis_lift.rActualPosSet	:= rPos_lift_up;
		st_mcAxis_lift.rVelocitySet	:= rVelocity_percent*200;
		st_mcAxis_bag.mcMoveAbsolute.Execute	:= TRUE;						
		st_mcAxis_bag.rActualPosSet	:= rPos_bag_closed;
		st_mcAxis_bag.rVelocitySet	:= rVelocity_percent*50;		
		roller_inbound.roller.forward	:= TRUE;
		roller_outbound.roller.forward	:= TRUE;
		roller_outbound_assist.roller.forward	:= TRUE;		
		valve_lift.extend 		:= TRUE;
		valve_lift.retract		:= FALSE;
		IF st_mcAxis_lift.mcMoveAbsolute.Done AND st_mcAxis_bag.mcMoveAbsolute.Done AND ton_aging_test.Q THEN
			st_mcAxis_lift.mcMoveAbsolute.Execute	:= FALSE;
			st_mcAxis_bag.mcMoveAbsolute.Execute	:= FALSE;
			roller_inbound.roller.forward	:= FALSE;
			roller_outbound.roller.forward	:= FALSE;
			roller_outbound_assist.roller.forward	:= FALSE;			
			ton_aging_test.IN	:= FALSE;			
			iAging_test	:= 2;
		END_IF	
	2:	
		ton_aging_test.PT	:= T#2S;
		ton_aging_test.IN	:= TRUE;
		IF ton_aging_test.Q THEN
			ton_aging_test.IN	:= FALSE;
			iAging_test	:= 3;				
		END_IF
	3://run backward
		ton_aging_test.PT	:= T#5S;
		ton_aging_test.IN	:= TRUE;
		st_mcAxis_lift.mcMoveAbsolute.Execute	:= TRUE;						
		st_mcAxis_lift.rActualPosSet	:= rPos_lift_down;
		st_mcAxis_lift.rVelocitySet	:= rVelocity_percent*200;
		st_mcAxis_bag.mcMoveAbsolute.Execute	:= TRUE;						
		st_mcAxis_bag.rActualPosSet	:= rPos_bag_opened;
		st_mcAxis_bag.rVelocitySet	:= rVelocity_percent*50;		
		roller_inbound.roller.forward	:= TRUE;
		roller_inbound.roller.backward	:= TRUE;
		roller_outbound.roller.backward	:= TRUE;
		roller_outbound_assist.roller.forward	:= TRUE;
		roller_outbound_assist.roller.backward	:= TRUE;
		
		valve_lift.extend 		:= FALSE;
		valve_lift.retract		:= TRUE;
		IF st_mcAxis_lift.mcMoveAbsolute.Done AND st_mcAxis_bag.mcMoveAbsolute.Done AND ton_aging_test.Q THEN
			st_mcAxis_lift.mcMoveAbsolute.Execute	:= FALSE;
			st_mcAxis_bag.mcMoveAbsolute.Execute	:= FALSE;
			roller_inbound.roller.forward	:= FALSE;
			roller_inbound.roller.backward	:= FALSE;
			roller_outbound.roller.backward	:= FALSE;
			roller_outbound_assist.roller.forward	:= FALSE;
			roller_outbound_assist.roller.backward	:= FALSE;		
			ton_aging_test.IN	:= FALSE;			
			iAging_test	:= 4;
		END_IF	
	4:
		ton_aging_test.PT	:= T#2S;
		ton_aging_test.IN	:= TRUE;
		IF ton_aging_test.Q THEN
			diCnt_aging	:= diCnt_aging+1;
			ton_aging_test.IN	:= FALSE;
			ADSLOGSTR(msgCtrlMask:=Tc2_System.ADSLOG_MSGTYPE_LOG,msgFmtStr:=CONCAT(STR1:=sInstanceName,STR2:=DINT_TO_STRING(diCnt_aging)),strArg:='');
			iAging_test	:= 1;				
		END_IF
	
		
		
		
	10://stop
		st_mcAxis_lift.mcMoveAbsolute.Execute	:= FALSE;
		st_mcAxis_bag.mcMoveAbsolute.Execute	:= FALSE;
		roller_inbound.roller.forward	:= FALSE;
		roller_outbound.roller.forward	:= FALSE;
		roller_outbound_assist.roller.forward	:= FALSE;		
		roller_inbound.roller.backward	:= FALSE;
		roller_outbound.roller.backward	:= FALSE;
		roller_outbound_assist.roller.backward	:= FALSE;	
		valve_lift.extend 		:= FALSE;
		valve_lift.retract		:= TRUE;
		ton_aging_test.IN	:= FALSE;	
		iAging_test	:= 0;

	END_CASE
END_METHOD

METHOD M_checkCondition : BOOL
VAR_INPUT
	condition	: E_Condition;
END_VAR

M_checkCondition	:= FALSE;
CASE condition OF
	E_Condition.NO_TOTE:
	 	IF NOT roller_inbound.photo_sensor[0].Q 
				OR NOT roller_inbound.photo_sensor[1].Q 
		THEN
			M_checkCondition	:= TRUE;
		END_IF
	E_Condition.TOTE_IN:
	 	IF  NOT roller_inbound.photo_sensor[0].Q
			AND  roller_inbound.photo_sensor[1].Q 
		THEN
			M_checkCondition	:= TRUE;
		END_IF	
	
	E_Condition.READY_LOADING_TOTE:
		//
		
	E_Condition.TOTE_READY:
		IF  ABS(AxisRef_lift.NcToPlc.ActPos-rPos_lift_down)<1 AND
			ABS(AxisRef_bag.NcToPlc.ActPos-rPos_bag_opened)<1 AND
			roller_inbound.photo_sensor[1].Q AND 
			photo_sensor_tote_detection.Q AND
			NOT roller_inbound.photo_sensor[0].Q AND 
			NOT roller_outbound.photo_sensor.Q AND
			valve_lift.retracted (*AND
			bag_opening_status_0.bag_status = BagStatus.OPENED AND 
			bag_opening_status_1._bagStatus = BagStatus.OPENED *)
		THEN
			tote_status	:= ToteStatus.LOADED;		
		ELSE
			IF tote_status = ToteStatus.LOADED THEN
				tote_status	:= ToteStatus.INBOUNDING;
			END_IF
		END_IF
		
		IF ABS(AxisRef_lift.NcToPlc.ActPos-rPos_lift_up)<1  
			AND NOT photo_sensor_tote_detection.Q
			AND NOT roller_inbound.photo_sensor[0].Q AND NOT roller_inbound.photo_sensor[1].Q 
			AND NOT roller_outbound.photo_sensor.Q AND valve_lift.retracted 
		THEN
			tote_status	:= ToteStatus.VACANT;	
		END_IF	
		
		IF NOT roller_inbound.photo_sensor[0].Q AND roller_inbound.photo_sensor[1].Q 
			AND photo_sensor_tote_detection.Q AND NOT roller_outbound.photo_sensor.Q 
		THEN
			IF tote_status=ToteStatus.VACANT THEN
				tote_status	:= ToteStatus.INBOUNDING;
			END_IF
		END_IF		

		M_checkCondition	:= TRUE;
END_CASE
END_METHOD

{attribute 'object_name' := 'M_Completing'}
METHOD M_Completing
CASE fbUnitModeManager.eModeStatus OF
	ePMLProtUnitMode_Production:
		;
END_CASE
END_METHOD

{attribute 'object_name' := 'M_Execute'}
METHOD M_Execute
CASE fbUnitModeManager.eModeStatus OF
	ePMLProtUnitMode_Production:		//Mode Production
		
//////////////////////////unloading///////////////////////	
				IF xOutbound THEN	
					IF M_unload() THEN
					 	xOutbound := FALSE;
					END_IF		
					RETURN;
				END_IF	
//////////////////////////loading///////////////////////
				IF xInbound THEN	
					IF M_load() THEN
						xInbound := FALSE;
					END_IF
				END_IF	

				
	ePMLProtUnitMode_Maintenance, ePMLUnitMode_Service:		
		;
	ePMLProtUnitMode_Manual:		//Manaul
	
END_CASE
END_METHOD

{attribute 'object_name' := 'M_Holding'}
METHOD M_Holding
CASE fbUnitModeManager.eModeStatus OF
	ePMLProtUnitMode_Production:		//Mode Production
		//Finisch the actual seperationstep	
		

	ePMLProtUnitMode_Maintenance:
		M_StateComplete();
END_CASE
END_METHOD

{attribute 'object_name' := 'M_Idle'}
METHOD M_Idle
ftrig_agingTest(CLK	:= bAging_test);
IF 	ftrig_agingTest.Q THEN
	iAging_test	:= 10;
END_IF
IF bAging_test THEN
	IF iAging_test=0 THEN
		iAging_test	:= 1;
	END_IF	
END_IF
M_agingTest(0.8);
END_METHOD

METHOD  M_load : BOOL
VAR_INPUT
END_VAR

VAR
	
END_VAR
M_load := FALSE;

//////////////////////////////////////////////////////////timeout//////////////////////////////////////////
		iStateTemp	:= eStateTemp;
//		ton_timeout();
		IF eStateTemp=eStates THEN
			ton_timeout.IN	:=TRUE;
		ELSE
			ton_timeout.IN	:=FALSE;
			eStateTemp	:= eStates;	
			M_Log(eLogType:=ServerityLevelType.INFO,sTextLog:='');
			IF ton_timeout.Q THEN
				RETURN;
			END_IF
		END_IF
		IF ton_timeout.Q THEN	
			ton_timeout.IN	:=FALSE;
			CASE eStates OF	
				E_LoadingStates.ERROR:	
					alarm_temp.Message	:= GenerateErrorMsg(errorType:='M',iState := iStateTemp,errorMsg:='in error state.');
				ELSE
					alarm_temp.Message	:= GenerateErrorMsg(errorType:='M',iState := iStateTemp,errorMsg:='time out');
			END_CASE
//////////////////////////////////////////////////////////states don't want to timeout and trig error//////////////////////////////////////////				
			IF  eStates<>E_WorkingStates.IDLE AND
				eStates<>E_WorkingStates.WAIT_NEW_TOTE AND
				eStates<>E_WorkingStates.WAIT AND
				eStates<>E_WorkingStates.BAG_OPEN_DETECTION AND
				eStates<>E_WorkingStates.WAIT_1 
			THEN
				tote_status	:= ToteStatus.MECHANICAL_ERROR;
				IF sInstanceName='working1' THEN					
					THIS^.pml_adminAlarm.M_SetAlarm(stAdmin:=GVL.PackTags1.Admin,stAlarm:=THIS^.alarm_temp);
				END_IF			
				IF sInstanceName='working2' THEN
					THIS^.pml_adminAlarm.M_SetAlarm(stAdmin:=GVL.PackTags2.Admin,stAlarm:=THIS^.alarm_temp);
				END_IF					
			END_IF
		END_IF
//////////////////////////////////////////////////////////conditions//////////////////////////////////////////

//////////////////////////////////////////////////////////excute//////////////////////////////////////////
CASE eStates OF 
		E_WorkingStates.IDLE:
			tote_status	:= ToteStatus.UNKNOWN;
//			xLoading	:= TRUE;
//			ton_timeout.PT	:= T#20MS;		
			st_mcAxis_lift.mcPower.Enable	:= TRUE;
			st_mcAxis_bag.mcPower.Enable	:= TRUE;
			st_mcAxis_lift.mcReset.Execute	:= TRUE;
			st_mcAxis_bag.mcReset.Execute	:= TRUE;
			IF st_mcAxis_lift.mcReadStatus.StandStill AND st_mcAxis_bag.mcReadStatus.StandStill  THEN
				eStates	:= E_WorkingStates.INIT;
			END_IF

		E_WorkingStates.INIT:
//			ADSLOGSTR(msgCtrlMask:= ADSLOG_MSGTYPE_LOG,msgFmtStr:='load start',strArg:='');
			ton_timeout.PT	:= T#3S;		
			st_mcAxis_lift.mcMoveAbsolute.Execute	:= FALSE;
			st_mcAxis_bag.mcMoveAbsolute.Execute	:= FALSE;			
			IF M_checkCondition(condition:=E_Condition.TOTE_READY) THEN///////////avoid recieve load signal from app many times
				IF tote_status=ToteStatus.LOADED  THEN
					IF sInstanceName='working1' THEN
						eStates	:= E_WorkingStates.DONE;
					END_IF
					IF sInstanceName='working2' THEN
						eStates	:= E_WorkingStates.DONE;
					END_IF					
				ELSE
					bagOpen_Status	:= bagOpenInit_Status;
					tote_status	:= ToteStatus.VACANT;					
					strLog_bagopen_detection	:= '';
					eStates	:= E_WorkingStates.BAG_OPEN_UP;
				END_IF
			END_IF		

		E_WorkingStates.BAG_OPEN_UP:	
			st_mcAxis_lift.mcMoveAbsolute.Execute	:= TRUE;		
			st_mcAxis_lift.rActualPosSet	:= rPos_lift_up;
			st_mcAxis_lift.rVelocitySet	:= 250;
			IF st_mcAxis_lift.mcMoveAbsolute.Done THEN
				st_mcAxis_lift.mcMoveAbsolute.Execute	:= FALSE;
				eStates	:= E_WorkingStates.BAG_OPEN_INIT;
			END_IF		
		E_WorkingStates.BAG_OPEN_INIT:	
			st_mcAxis_bag.mcMoveAbsolute.Execute	:= TRUE;
			st_mcAxis_bag.rVelocitySet	:= 250;
			IF bUsingOpenBag THEN
				st_mcAxis_bag.rActualPosSet	:= rPos_bag_closed;
			ELSE
				st_mcAxis_bag.rActualPosSet	:= rPos_bag_opened;
			END_IF
			IF st_mcAxis_bag.mcMoveAbsolute.Done THEN
				st_mcAxis_bag.bTouchTorque := FALSE;
				st_mcAxis_bag.mcMoveAbsolute.Execute	:= FALSE;
				eStates	:= E_WorkingStates.TOTE_LIFT_DOWN;
			END_IF				
			
		E_WorkingStates.TOTE_LIFT_DOWN:			
			valve_lift.extend	:= FALSE;
			valve_lift.retract	:= TRUE;
			IF NOT valve_lift.extended AND valve_lift.retracted THEN
				eStates	:= E_WorkingStates.WAIT_NEW_TOTE;
			END_IF	
			
